C03657=1192.781,332.000,-73.266,-176.346,7.864,148.456
C03658=1192.786,331.751,-73.233,-176.349,7.861,148.456
C03659=1192.790,331.504,-73.202,-176.351,7.857,148.456
C03660=1192.794,331.256,-73.170,-176.354,7.854,148.456
C03661=1192.798,331.008,-73.138,-176.356,7.851,148.455
C03662=1192.803,330.759,-73.107,-176.358,7.849,148.456
C03663=1192.807,330.511,-73.075,-176.360,7.845,148.455
C03664=1192.811,330.264,-73.043,-176.363,7.842,148.455
C03665=1192.815,330.016,-73.011,-176.365,7.839,148.455
C03666=1192.819,329.768,-72.979,-176.367,7.836,148.455
C03667=1192.823,329.520,-72.948,-176.370,7.834,148.455
C03668=1192.827,329.272,-72.916,-176.372,7.830,148.455
C03669=1192.832,329.023,-72.884,-176.375,7.827,148.455
C03670=1192.836,328.776,-72.853,-176.377,7.824,148.455
C03671=1192.840,328.528,-72.821,-176.379,7.821,148.454
C03672=1192.844,328.281,-72.789,-176.382,7.818,148.454
C03673=1192.848,328.033,-72.757,-176.383,7.815,148.454
C03674=1192.853,327.784,-72.726,-176.386,7.812,148.454
C03675=1192.857,327.536,-72.694,-176.388,7.809,148.454
C03676=1192.861,327.288,-72.662,-176.391,7.806,148.454
C03677=1192.865,327.040,-72.632,-176.393,7.802,148.454
C03678=1192.869,326.792,-72.600,-176.395,7.800,148.454
C03679=1192.873,326.545,-72.568,-176.398,7.797,148.454
C03680=1192.878,326.296,-72.537,-176.400,7.794,148.454
C03681=1192.882,326.049,-72.505,-176.403,7.791,148.453
C03682=1192.886,325.801,-72.473,-176.405,7.788,148.453
C03683=1192.891,325.553,-72.443,-176.407,7.785,148.453
C03684=1192.894,325.305,-72.411,-176.410,7.782,148.453
C03685=1192.899,325.057,-72.379,-176.412,7.779,148.453
C03686=1192.903,324.809,-72.348,-176.415,7.776,148.453
C03687=1192.906,324.561,-72.316,-176.417,7.772,148.453
C03688=1192.911,324.313,-72.285,-176.419,7.770,148.453
C03689=1192.915,324.064,-72.253,-176.421,7.767,148.453
C03690=1192.920,323.817,-72.222,-176.424,7.764,148.453
C03691=1192.924,323.568,-72.190,-176.427,7.761,148.453
C03692=1192.928,323.321,-72.159,-176.429,7.757,148.452
C03693=1192.932,323.072,-72.128,-176.432,7.754,148.452
C03694=1192.936,322.825,-72.096,-176.433,7.752,148.452
C03695=1192.940,322.576,-72.065,-176.436,7.749,148.452
C03696=1192.945,322.329,-72.034,-176.438,7.746,148.452
C03697=1192.949,322.081,-72.003,-176.441,7.743,148.452
C03698=1192.953,321.832,-71.972,-176.444,7.740,148.452
C03699=1192.958,321.585,-71.940,-176.445,7.737,148.452
C03700=1192.962,321.336,-71.909,-176.448,7.734,148.452
C03701=1192.966,321.089,-71.878,-176.450,7.731,148.452
C03702=1192.970,320.840,-71.847,-176.453,7.728,148.452
C03703=1192.974,320.593,-71.815,-176.455,7.726,148.452
C03704=1192.978,320.344,-71.784,-176.457,7.722,148.452
C03705=1192.982,320.097,-71.754,-176.460,7.719,148.452
C03706=1192.986,319.849,-71.722,-176.462,7.716,148.451
C03707=1192.990,319.601,-71.691,-176.465,7.713,148.451
C03708=1192.995,319.353,-71.660,-176.467,7.711,148.451
C03709=1192.999,319.105,-71.629,-176.469,7.707,148.451
C03710=1193.003,318.857,-71.598,-176.472,7.704,148.451
C03711=1193.007,318.608,-71.567,-176.475,7.701,148.451
C03712=1193.012,318.360,-71.536,-176.477,7.698,148.451
C03713=1193.016,318.113,-71.504,-176.479,7.696,148.451
C03714=1193.020,317.864,-71.473,-176.482,7.693,148.451
C03715=1193.024,317.616,-71.443,-176.484,7.689,148.451
C03716=1193.029,317.369,-71.412,-176.487,7.686,148.451
C03717=1193.033,317.120,-71.381,-176.489,7.683,148.451
C03718=1193.037,316.873,-71.350,-176.491,7.681,148.451
C03719=1193.041,316.624,-71.319,-176.494,7.678,148.451
C03720=1193.046,316.376,-71.288,-176.496,7.675,148.451
C03721=1193.050,316.128,-71.258,-176.499,7.672,148.451
C03722=1193.054,315.880,-71.227,-176.501,7.669,148.451
C03723=1193.058,315.632,-71.195,-176.504,7.666,148.451
C03724=1193.063,315.384,-71.164,-176.506,7.663,148.450
C03725=1193.067,315.136,-71.133,-176.508,7.660,148.450
C03726=1193.072,314.859,-71.100,-176.511,7.657,148.450
C03727=1193.076,314.583,-71.065,-176.514,7.654,148.450
C03728=1193.081,314.307,-71.031,-176.517,7.651,148.450
C03729=1193.085,314.030,-70.997,-176.519,7.647,148.450
C03730=1193.090,313.782,-70.966,-176.522,7.645,148.450
C03731=1193.094,313.534,-70.935,-176.524,7.642,148.450
C03732=1193.098,313.286,-70.905,-176.527,7.639,148.450
C03733=1193.102,313.038,-70.874,-176.529,7.635,148.450
C03734=1193.107,312.790,-70.843,-176.531,7.633,148.450
C03735=1193.111,312.542,-70.812,-176.534,7.630,148.450
C03736=1193.115,312.293,-70.782,-176.537,7.627,148.450
C03737=1193.119,312.045,-70.751,-176.539,7.624,148.450
C03738=1193.124,311.797,-70.720,-176.542,7.621,148.450
C03739=1193.128,311.550,-70.690,-176.544,7.619,148.450
C03740=1193.132,311.301,-70.659,-176.546,7.616,148.450
C03741=1193.136,311.053,-70.628,-176.549,7.612,148.450
C03742=1193.140,310.805,-70.598,-176.551,7.609,148.450
C03743=1193.145,310.558,-70.567,-176.554,7.607,148.450
C03744=1193.149,310.309,-70.538,-176.556,7.604,148.450
C03745=1193.153,310.061,-70.507,-176.559,7.601,148.450
C03746=1193.158,309.813,-70.476,-176.561,7.598,148.450
C03747=1193.162,309.565,-70.446,-176.563,7.596,148.450
C03748=1193.166,309.317,-70.415,-176.566,7.593,148.450
C03749=1193.170,309.068,-70.384,-176.569,7.590,148.450
C03750=1193.174,308.820,-70.355,-176.571,7.586,148.450
C03751=1193.179,308.572,-70.324,-176.573,7.584,148.450
C03752=1193.183,308.325,-70.294,-176.576,7.581,148.450
C03753=1193.188,308.077,-70.263,-176.579,7.578,148.450
C03754=1193.191,307.828,-70.233,-176.581,7.575,148.450
C03755=1193.196,307.580,-70.202,-176.583,7.573,148.450
C03756=1193.200,307.332,-70.172,-176.586,7.569,148.450
C03757=1193.205,307.083,-70.142,-176.588,7.566,148.450
C03758=1193.208,306.836,-70.112,-176.591,7.563,148.450
C03759=1193.213,306.588,-70.081,-176.593,7.561,148.450
C03760=1193.217,306.339,-70.051,-176.596,7.558,148.450
C03761=1193.221,306.091,-70.021,-176.599,7.555,148.450
C03762=1193.225,305.843,-69.990,-176.601,7.552,148.449
C03763=1193.230,305.595,-69.960,-176.603,7.550,148.449
C03764=1193.234,305.347,-69.930,-176.606,7.547,148.450
C03765=1193.239,305.098,-69.900,-176.608,7.544,148.450
C03766=1193.243,304.851,-69.870,-176.611,7.541,148.450
C03767=1193.247,304.603,-69.839,-176.613,7.539,148.450
C03768=1193.251,304.354,-69.809,-176.616,7.536,148.450
C03769=1193.255,304.106,-69.779,-176.618,7.532,148.449
C03770=1193.260,303.858,-69.749,-176.621,7.529,148.449
C03771=1193.264,303.610,-69.719,-176.623,7.527,148.450
C03772=1193.268,303.361,-69.689,-176.626,7.524,148.450
C03773=1193.272,303.114,-69.659,-176.628,7.521,148.450
C03774=1193.277,302.865,-69.629,-176.631,7.518,148.450
C03775=1193.281,302.618,-69.599,-176.633,7.516,148.450
C03776=1193.285,302.369,-69.569,-176.636,7.513,148.450
C03777=1193.290,302.121,-69.539,-176.639,7.510,148.450
C03778=1193.294,301.873,-69.509,-176.640,7.507,148.450
C03779=1193.298,301.625,-69.479,-176.643,7.504,148.450
C03780=1193.303,301.377,-69.449,-176.646,7.501,148.450
C03781=1193.306,301.128,-69.419,-176.648,7.498,148.450
C03782=1193.311,300.880,-69.389,-176.651,7.496,148.450
C03783=1193.315,300.632,-69.359,-176.653,7.493,148.450
C03784=1193.319,300.383,-69.329,-176.656,7.490,148.450
C03785=1193.324,300.135,-69.300,-176.658,7.488,148.450
C03786=1193.328,299.887,-69.269,-176.661,7.485,148.450
C03787=1193.332,299.639,-69.239,-176.664,7.482,148.450
C03788=1193.337,299.391,-69.210,-176.666,7.479,148.450
C03789=1193.340,299.143,-69.180,-176.668,7.477,148.450
C03790=1193.345,298.894,-69.150,-176.671,7.473,148.450
C03791=1193.350,298.646,-69.120,-176.673,7.470,148.450
C03792=1193.354,298.398,-69.091,-176.676,7.468,148.450
C03793=1193.358,298.150,-69.061,-176.678,7.465,148.450
C03794=1193.363,297.902,-69.031,-176.681,7.462,148.450
C03795=1193.367,297.653,-69.001,-176.684,7.459,148.450
C03796=1193.371,297.405,-68.972,-176.686,7.457,148.450
C03797=1193.375,297.157,-68.942,-176.688,7.454,148.450
C03798=1193.379,296.909,-68.912,-176.691,7.451,148.450
C03799=1193.384,296.661,-68.882,-176.693,7.449,148.450
C03800=1193.388,296.412,-68.853,-176.696,7.446,148.450
C03801=1193.392,296.164,-68.823,-176.699,7.443,148.450
C03802=1193.396,295.916,-68.794,-176.701,7.441,148.450
C03803=1193.401,295.668,-68.765,-176.704,7.438,148.450
C03804=1193.405,295.420,-68.735,-176.706,7.435,148.450
C03805=1193.410,295.172,-68.706,-176.709,7.432,148.450
C03806=1193.414,294.924,-68.675,-176.711,7.429,148.450
C03807=1193.418,294.675,-68.646,-176.714,7.426,148.450
C03808=1193.423,294.427,-68.616,-176.717,7.423,148.450
C03809=1193.427,294.179,-68.587,-176.719,7.421,148.450
C03810=1193.431,293.931,-68.557,-176.721,7.418,148.450
C03811=1193.435,293.682,-68.528,-176.724,7.415,148.450
C03812=1193.439,293.434,-68.498,-176.726,7.413,148.450
C03813=1193.443,293.186,-68.469,-176.729,7.410,148.450
C03814=1193.448,292.938,-68.439,-176.732,7.407,148.450
C03815=1193.452,292.690,-68.410,-176.734,7.405,148.451
C03816=1193.457,292.442,-68.381,-176.737,7.402,148.451
C03817=1193.461,292.193,-68.352,-176.739,7.399,148.451
C03818=1193.465,291.945,-68.323,-176.741,7.397,148.451
C03819=1193.469,291.696,-68.293,-176.744,7.394,148.451
C03820=1193.474,291.448,-68.264,-176.747,7.391,148.451
C03821=1193.478,291.200,-68.234,-176.749,7.388,148.451
C03822=1193.482,290.952,-68.205,-176.752,7.385,148.451
C03823=1193.487,290.704,-68.176,-176.754,7.382,148.451
C03824=1193.491,290.456,-68.146,-176.757,7.380,148.451
C03825=1193.495,290.207,-68.118,-176.759,7.377,148.451
C03826=1193.500,289.959,-68.088,-176.762,7.374,148.451
C03827=1193.504,289.710,-68.059,-176.764,7.372,148.451
C03828=1193.508,289.462,-68.029,-176.767,7.369,148.451
C03829=1193.513,289.214,-68.000,-176.769,7.366,148.451
C03830=1193.517,288.939,-67.968,-176.773,7.363,148.451
C03831=1193.523,288.665,-67.936,-176.775,7.360,148.451
C03832=1193.527,288.391,-67.903,-176.778,7.357,148.451
C03833=1193.531,288.116,-67.871,-176.781,7.354,148.451
C03834=1193.536,287.868,-67.842,-176.784,7.351,148.451
C03835=1193.541,287.619,-67.814,-176.786,7.349,148.452
C03836=1193.545,287.371,-67.784,-176.788,7.346,148.452
C03837=1193.549,287.123,-67.755,-176.791,7.343,148.452
C03838=1193.554,286.875,-67.726,-176.793,7.341,148.452
C03839=1193.558,286.626,-67.697,-176.796,7.338,148.452
C03840=1193.562,286.378,-67.668,-176.799,7.336,148.452
C03841=1193.566,286.130,-67.639,-176.801,7.333,148.452
C03842=1193.570,285.881,-67.610,-176.804,7.330,148.452
C03843=1193.575,285.634,-67.581,-176.806,7.328,148.452
C03844=1193.580,285.385,-67.552,-176.809,7.325,148.452
C03845=1193.584,285.137,-67.523,-176.812,7.322,148.452
C03846=1193.588,284.889,-67.495,-176.814,7.320,148.452
C03847=1193.592,284.640,-67.465,-176.816,7.317,148.452
C03848=1193.597,284.392,-67.437,-176.819,7.314,148.452
C03849=1193.601,284.143,-67.407,-176.821,7.311,148.452
C03850=1193.605,283.895,-67.379,-176.824,7.309,148.453
C03851=1193.609,283.647,-67.350,-176.827,7.307,148.453
C03852=1193.614,283.398,-67.321,-176.829,7.304,148.453
C03853=1193.619,283.151,-67.292,-176.832,7.301,148.453
C03854=1193.622,282.902,-67.264,-176.834,7.298,148.453
C03855=1193.627,282.654,-67.235,-176.837,7.295,148.453
C03856=1193.632,282.406,-67.206,-176.840,7.292,148.453
C03857=1193.636,282.157,-67.177,-176.842,7.290,148.453
C03858=1193.640,281.909,-67.149,-176.844,7.287,148.453
C03859=1193.645,281.661,-67.120,-176.847,7.285,148.453
C03860=1193.649,281.412,-67.091,-176.850,7.282,148.453
C03861=1193.653,281.164,-67.063,-176.852,7.279,148.453
C03862=1193.657,280.916,-67.033,-176.855,7.277,148.453
C03863=1193.662,280.667,-67.005,-176.857,7.274,148.453
C03864=1193.666,280.419,-66.977,-176.859,7.272,148.454
C03865=1193.670,280.171,-66.948,-176.862,7.269,148.454
C03866=1193.674,279.923,-66.919,-176.865,7.266,148.454
C03867=1193.679,279.674,-66.891,-176.868,7.264,148.454
C03868=1193.684,279.426,-66.862,-176.870,7.261,148.454
C03869=1193.687,279.178,-66.833,-176.872,7.259,148.454
C03870=1193.692,278.929,-66.805,-176.875,7.256,148.454
C03871=1193.696,278.681,-66.777,-176.878,7.253,148.454
C03872=1193.700,278.433,-66.747,-176.880,7.251,148.454
C03873=1193.705,278.184,-66.719,-176.883,7.248,148.454
C03874=1193.709,277.936,-66.691,-176.885,7.246,148.454
C03875=1193.714,277.688,-66.663,-176.888,7.243,148.455
C03876=1193.718,277.439,-66.634,-176.891,7.240,148.455
C03877=1193.722,277.191,-66.605,-176.893,7.238,148.455
C03878=1193.726,276.943,-66.577,-176.896,7.235,148.455
C03879=1193.731,276.694,-66.548,-176.898,7.233,148.455
C03880=1193.735,276.446,-66.521,-176.901,7.230,148.455
C03881=1193.740,276.197,-66.492,-176.904,7.227,148.455
C03882=1193.744,275.949,-66.464,-176.906,7.225,148.455
C03883=1193.749,275.700,-66.435,-176.909,7.222,148.455
C03884=1193.752,275.452,-66.407,-176.911,7.220,148.455
C03885=1193.757,275.204,-66.379,-176.914,7.217,148.455
C03886=1193.761,274.956,-66.350,-176.916,7.215,148.456
C03887=1193.766,274.708,-66.322,-176.919,7.212,148.456
C03888=1193.770,274.459,-66.294,-176.921,7.209,148.456
C03889=1193.775,274.211,-66.265,-176.924,7.207,148.456
C03890=1193.779,273.962,-66.237,-176.927,7.204,148.456
C03891=1193.783,273.714,-66.209,-176.929,7.202,148.456
C03892=1193.787,273.465,-66.181,-176.932,7.199,148.456
C03893=1193.792,273.218,-66.153,-176.934,7.197,148.456
C03894=1193.796,272.969,-66.124,-176.937,7.194,148.456
C03895=1193.801,272.721,-66.096,-176.940,7.191,148.456
C03896=1193.805,272.472,-66.069,-176.942,7.189,148.457
C03897=1193.810,272.223,-66.040,-176.944,7.186,148.457
C03898=1193.814,271.975,-66.012,-176.947,7.184,148.457
C03899=1193.819,271.727,-65.984,-176.950,7.181,148.457
C03900=1193.822,271.478,-65.956,-176.952,7.179,148.457
C03901=1193.827,271.230,-65.928,-176.955,7.176,148.457
C03902=1193.831,270.981,-65.899,-176.957,7.174,148.457
C03903=1193.836,270.733,-65.871,-176.960,7.171,148.457
C03904=1193.840,270.486,-65.844,-176.962,7.169,148.457
C03905=1193.845,270.236,-65.816,-176.965,7.166,148.458
C03906=1193.849,269.988,-65.788,-176.968,7.163,148.458
C03907=1193.853,269.740,-65.760,-176.970,7.161,148.458
C03908=1193.858,269.491,-65.731,-176.973,7.158,148.458
C03909=1193.862,269.243,-65.703,-176.975,7.156,148.458
C03910=1193.866,268.994,-65.676,-176.978,7.153,148.458
C03911=1193.871,268.747,-65.648,-176.980,7.151,148.458
C03912=1193.875,268.498,-65.620,-176.983,7.148,148.458
C03913=1193.879,268.250,-65.592,-176.985,7.146,148.458
C03914=1193.884,268.001,-65.564,-176.988,7.143,148.459
C03915=1193.888,267.753,-65.537,-176.991,7.141,148.459
C03916=1193.893,267.504,-65.508,-176.993,7.138,148.459
C03917=1193.897,267.255,-65.481,-176.995,7.136,148.459
C03918=1193.901,267.007,-65.453,-176.999,7.133,148.459
C03919=1193.905,266.759,-65.425,-177.001,7.131,148.459
C03920=1193.910,266.510,-65.398,-177.004,7.128,148.459
C03921=1193.915,266.262,-65.370,-177.006,7.126,148.460
C03922=1193.919,266.014,-65.341,-177.009,7.123,148.460
C03923=1193.923,265.765,-65.314,-177.011,7.121,148.460
C03924=1193.928,265.517,-65.287,-177.014,7.118,148.460
C03925=1193.932,265.268,-65.259,-177.016,7.116,148.460
C03926=1193.936,265.020,-65.231,-177.019,7.113,148.460
C03927=1193.941,264.771,-65.204,-177.021,7.111,148.460
C03928=1193.945,264.523,-65.176,-177.024,7.108,148.460
C03929=1193.950,264.275,-65.148,-177.027,7.106,148.461
C03930=1193.954,264.026,-65.121,-177.029,7.103,148.461
C03931=1193.958,263.778,-65.093,-177.031,7.101,148.461
C03932=1193.963,263.529,-65.065,-177.035,7.098,148.461
C03933=1193.967,263.281,-65.038,-177.037,7.096,148.461
C03934=1193.972,263.007,-65.008,-177.040,7.093,148.461
C03935=1193.977,262.735,-64.977,-177.043,7.090,148.461
C03936=1193.982,262.463,-64.948,-177.045,7.087,148.461
C03937=1193.986,262.189,-64.917,-177.049,7.085,148.462
C03938=1193.991,261.941,-64.889,-177.051,7.082,148.462
C03939=1193.995,261.693,-64.862,-177.054,7.080,148.462
C03940=1193.999,261.444,-64.834,-177.056,7.078,148.462
C03941=1194.004,261.196,-64.807,-177.059,7.075,148.462
C03942=1194.008,260.947,-64.780,-177.061,7.073,148.462
C03943=1194.013,260.699,-64.752,-177.064,7.070,148.462
C03944=1194.017,260.450,-64.725,-177.066,7.068,148.463
C03945=1194.022,260.202,-64.698,-177.070,7.065,148.463
C03946=1194.026,259.954,-64.670,-177.072,7.063,148.463
C03947=1194.031,259.705,-64.643,-177.074,7.060,148.463
C03948=1194.035,259.456,-64.615,-177.077,7.058,148.463
C03949=1194.039,259.208,-64.588,-177.079,7.056,148.463
C03950=1194.044,258.960,-64.561,-177.082,7.053,148.463
C03951=1194.048,258.711,-64.534,-177.085,7.051,148.464
C03952=1194.053,258.463,-64.506,-177.087,7.048,148.464
C03953=1194.057,258.214,-64.478,-177.089,7.046,148.464
C03954=1194.061,257.966,-64.451,-177.093,7.043,148.464
C03955=1194.066,257.717,-64.424,-177.095,7.041,148.464
C03956=1194.071,257.469,-64.397,-177.097,7.038,148.464
C03957=1194.075,257.220,-64.370,-177.100,7.036,148.465
C03958=1194.078,256.972,-64.343,-177.102,7.034,148.465
C03959=1194.083,256.723,-64.315,-177.105,7.031,148.465
C03960=1194.088,256.475,-64.288,-177.108,7.029,148.465
C03961=1194.092,256.226,-64.261,-177.110,7.026,148.465
C03962=1194.097,255.978,-64.234,-177.113,7.024,148.465
C03963=1194.102,255.729,-64.207,-177.116,7.021,148.465
C03964=1194.106,255.480,-64.180,-177.118,7.019,148.466
C03965=1194.110,255.232,-64.153,-177.121,7.016,148.466
C03966=1194.114,254.984,-64.126,-177.123,7.014,148.466
C03967=1194.119,254.736,-64.098,-177.126,7.012,148.466
C03968=1194.123,254.487,-64.071,-177.129,7.009,148.466
C03969=1194.128,254.239,-64.044,-177.131,7.007,148.466
C03970=1194.132,253.991,-64.018,-177.134,7.004,148.467
C03971=1194.136,253.741,-63.990,-177.136,7.002,148.467
C03972=1194.140,253.493,-63.963,-177.139,7.000,148.467
C03973=1194.145,253.244,-63.936,-177.141,6.997,148.467
C03974=1194.150,252.996,-63.909,-177.144,6.995,148.467
C03975=1194.154,252.748,-63.883,-177.147,6.993,148.467
C03976=1194.158,252.499,-63.856,-177.149,6.990,148.468
C03977=1194.163,252.251,-63.829,-177.152,6.988,148.468
C03978=1194.168,252.002,-63.802,-177.154,6.986,148.468
C03979=1194.172,251.753,-63.776,-177.156,6.983,148.468
C03980=1194.177,251.505,-63.749,-177.160,6.981,148.468
C03981=1194.181,251.256,-63.722,-177.162,6.979,148.468
C03982=1194.185,251.008,-63.695,-177.165,6.976,148.469
C03983=1194.189,250.759,-63.668,-177.167,6.974,148.469
C03984=1194.194,250.511,-63.641,-177.170,6.972,148.469
C03985=1194.198,250.262,-63.614,-177.172,6.969,148.469
C03986=1194.202,250.014,-63.587,-177.175,6.967,148.469
C03987=1194.207,249.765,-63.561,-177.178,6.964,148.469
C03988=1194.211,249.517,-63.534,-177.180,6.962,148.470
C03989=1194.216,249.268,-63.507,-177.183,6.960,148.470
C03990=1194.221,249.020,-63.480,-177.185,6.957,148.470
C03991=1194.225,248.771,-63.454,-177.188,6.955,148.470
C03992=1194.230,248.522,-63.428,-177.191,6.952,148.470
C03993=1194.234,248.274,-63.400,-177.193,6.950,148.471
C03994=1194.238,248.026,-63.374,-177.195,6.948,148.471
C03995=1194.243,247.777,-63.347,-177.199,6.946,148.471
C03996=1194.247,247.528,-63.321,-177.201,6.943,148.471
C03997=1194.252,247.280,-63.294,-177.204,6.940,148.471
C03998=1194.256,247.031,-63.267,-177.206,6.939,148.471
C03999=1194.261,246.782,-63.241,-177.208,6.936,148.472
C04000=1194.265,246.534,-63.214,-177.212,6.934,148.472
C04001=1194.269,246.286,-63.188,-177.214,6.932,148.472
C04002=1194.274,246.037,-63.161,-177.216,6.930,148.472
C04003=1194.278,245.788,-63.135,-177.219,6.927,148.472
C04004=1194.283,245.540,-63.108,-177.222,6.925,148.473
C04005=1194.287,245.291,-63.082,-177.224,6.923,148.473
C04006=1194.291,245.043,-63.055,-177.227,6.920,148.473
C04007=1194.296,244.794,-63.029,-177.229,6.918,148.473
C04008=1194.300,244.545,-63.002,-177.232,6.915,148.473
C04009=1194.305,244.298,-62.976,-177.235,6.913,148.473
C04010=1194.310,244.049,-62.950,-177.237,6.911,148.474
C04011=1194.314,243.801,-62.923,-177.240,6.908,148.474
C04012=1194.319,243.551,-62.897,-177.243,6.907,148.474
C04013=1194.323,243.303,-62.871,-177.245,6.904,148.474
C04014=1194.328,243.054,-62.844,-177.248,6.902,148.475
C04015=1194.332,242.806,-62.818,-177.250,6.900,148.475
C04016=1194.337,242.557,-62.791,-177.253,6.898,148.475
C04017=1194.340,242.309,-62.765,-177.255,6.895,148.475
C04018=1194.345,242.060,-62.739,-177.258,6.893,148.475
C04019=1194.349,241.811,-62.712,-177.260,6.891,148.475
C04020=1194.354,241.563,-62.687,-177.263,6.888,148.476
C04021=1194.359,241.314,-62.660,-177.266,6.886,148.476
C04022=1194.363,241.066,-62.634,-177.268,6.884,148.476
C04023=1194.367,240.817,-62.608,-177.271,6.881,148.476
C04024=1194.372,240.569,-62.581,-177.274,6.879,148.476
C04025=1194.376,240.320,-62.555,-177.276,6.877,148.477
C04026=1194.380,240.071,-62.530,-177.279,6.874,148.477
C04027=1194.385,239.823,-62.503,-177.281,6.872,148.477
C04028=1194.390,239.575,-62.477,-177.284,6.870,148.477
C04029=1194.394,239.326,-62.451,-177.287,6.868,148.478
C04030=1194.399,239.077,-62.424,-177.289,6.866,148.478
C04031=1194.403,238.828,-62.399,-177.292,6.864,148.478
C04032=1194.407,238.580,-62.373,-177.294,6.861,148.478
C04033=1194.412,238.332,-62.346,-177.297,6.859,148.478
C04034=1194.417,238.083,-62.320,-177.299,6.857,148.478
C04035=1194.421,237.834,-62.295,-177.302,6.854,148.479
C04036=1194.426,237.585,-62.268,-177.305,6.852,148.479
C04037=1194.430,237.337,-62.242,-177.307,6.850,148.479
C04038=1194.435,237.066,-62.214,-177.310,6.847,148.479
C04039=1194.440,236.794,-62.186,-177.313,6.845,148.480
C04040=1194.444,236.523,-62.157,-177.316,6.843,148.480
C04041=1194.450,236.250,-62.129,-177.319,6.840,148.480
C04042=1194.454,236.002,-62.103,-177.321,6.838,148.480
C04043=1194.458,235.754,-62.077,-177.324,6.836,148.481
C04044=1194.463,235.505,-62.051,-177.327,6.833,148.481
C04045=1194.467,235.256,-62.025,-177.329,6.831,148.481
C04046=1194.472,235.008,-61.999,-177.332,6.829,148.481
C04047=1194.477,234.759,-61.974,-177.334,6.827,148.481
C04048=1194.481,234.510,-61.948,-177.337,6.825,148.482
C04049=1194.485,234.262,-61.922,-177.339,6.822,148.482
C04050=1194.490,234.013,-61.897,-177.342,6.821,148.482
C04051=1194.495,233.764,-61.870,-177.345,6.818,148.482
C04052=1194.499,233.516,-61.844,-177.347,6.816,148.482
C04053=1194.503,233.267,-61.818,-177.350,6.814,148.483
C04054=1194.508,233.019,-61.793,-177.352,6.812,148.483
C04055=1194.512,232.770,-61.767,-177.355,6.809,148.483
C04056=1194.516,232.522,-61.741,-177.358,6.807,148.484
C04057=1194.521,232.274,-61.716,-177.360,6.805,148.484
C04058=1194.525,232.025,-61.690,-177.363,6.802,148.484
C04059=1194.530,231.776,-61.664,-177.366,6.800,148.484
C04060=1194.534,231.527,-61.638,-177.368,6.798,148.484
C04061=1194.540,231.278,-61.613,-177.371,6.797,148.485
C04062=1194.544,231.029,-61.588,-177.374,6.794,148.485
C04063=1194.548,230.780,-61.562,-177.376,6.792,148.485
C04064=1194.553,230.532,-61.537,-177.378,6.790,148.485
C04065=1194.557,230.284,-61.511,-177.381,6.788,148.486
C04066=1194.561,230.035,-61.485,-177.384,6.785,148.486
C04067=1194.566,229.787,-61.460,-177.386,6.783,148.486
C04068=1194.570,229.538,-61.434,-177.389,6.781,148.486
C04069=1194.575,229.289,-61.408,-177.392,6.779,148.487
C04070=1194.579,229.041,-61.383,-177.394,6.776,148.487
C04071=1194.584,228.792,-61.358,-177.397,6.775,148.487
C04072=1194.589,228.543,-61.332,-177.400,6.773,148.487
C04073=1194.593,228.295,-61.307,-177.402,6.770,148.487
C04074=1194.597,228.046,-61.281,-177.405,6.768,148.488
C04075=1194.602,227.798,-61.255,-177.407,6.766,148.488
C04076=1194.607,227.548,-61.230,-177.410,6.764,148.488
C04077=1194.611,227.299,-61.205,-177.413,6.762,148.488
C04078=1194.616,227.051,-61.179,-177.415,6.759,148.489
C04079=1194.620,226.803,-61.154,-177.418,6.757,148.489
C04080=1194.625,226.554,-61.129,-177.421,6.755,148.489
C04081=1194.629,226.305,-61.103,-177.423,6.753,148.489
C04082=1194.633,226.056,-61.077,-177.426,6.751,148.490
C04083=1194.638,225.808,-61.053,-177.429,6.749,148.490
C04084=1194.642,225.559,-61.028,-177.431,6.747,148.490
C04085=1194.647,225.311,-61.002,-177.433,6.745,148.490
C04086=1194.651,225.061,-60.977,-177.437,6.742,148.491
C04087=1194.656,224.813,-60.952,-177.439,6.740,148.491
C04088=1194.660,224.565,-60.926,-177.441,6.738,148.491
C04089=1194.666,224.316,-60.901,-177.444,6.736,148.491
C04090=1194.670,224.067,-60.876,-177.447,6.733,148.491
C04091=1194.674,223.818,-60.850,-177.449,6.732,148.492
C04092=1194.678,223.570,-60.826,-177.452,6.730,148.492
C04093=1194.683,223.321,-60.800,-177.455,6.728,148.492
C04094=1194.688,223.072,-60.775,-177.457,6.726,148.493
C04095=1194.692,222.824,-60.750,-177.460,6.723,148.493
C04096=1194.697,222.575,-60.725,-177.463,6.721,148.493
C04097=1194.701,222.326,-60.700,-177.465,6.719,148.493
C04098=1194.706,222.078,-60.675,-177.468,6.717,148.494
C04099=1194.710,221.829,-60.649,-177.471,6.715,148.494
C04100=1194.715,221.580,-60.625,-177.473,6.713,148.494
C04101=1194.719,221.331,-60.599,-177.476,6.711,148.494
C04102=1194.724,221.083,-60.575,-177.478,6.709,148.495
C04103=1194.728,220.834,-60.549,-177.481,6.707,148.495
C04104=1194.733,220.585,-60.524,-177.484,6.704,148.495
C04105=1194.737,220.336,-60.499,-177.486,6.702,148.495
C04106=1194.742,220.088,-60.475,-177.489,6.700,148.496
C04107=1194.746,219.839,-60.449,-177.491,6.698,148.496
C04108=1194.751,219.591,-60.424,-177.494,6.696,148.496
C04109=1194.755,219.341,-60.400,-177.497,6.694,148.497
C04110=1194.760,219.093,-60.374,-177.500,6.692,148.497
C04111=1194.765,218.845,-60.350,-177.502,6.690,148.497
C04112=1194.769,218.595,-60.325,-177.504,6.688,148.497
C04113=1194.773,218.347,-60.300,-177.507,6.686,148.498
C04114=1194.778,218.098,-60.275,-177.510,6.684,148.498
C04115=1194.783,217.849,-60.250,-177.512,6.681,148.498
C04116=1194.787,217.601,-60.225,-177.515,6.680,148.498
C04117=1194.792,217.352,-60.200,-177.518,6.678,148.499
C04118=1194.795,217.103,-60.176,-177.520,6.676,148.499
C04119=1194.800,216.855,-60.150,-177.523,6.673,148.499
C04120=1194.805,216.606,-60.126,-177.526,6.671,148.499
C04121=1194.809,216.357,-60.101,-177.528,6.669,148.500
C04122=1194.814,216.108,-60.077,-177.531,6.667,148.500
C04123=1194.819,215.859,-60.051,-177.533,6.665,148.500
C04124=1194.823,215.611,-60.027,-177.536,6.663,148.501
C04125=1194.828,215.362,-60.002,-177.539,6.661,148.501
C04126=1194.832,215.113,-59.978,-177.542,6.659,148.501
C04127=1194.837,214.864,-59.953,-177.544,6.657,148.501
C04128=1194.841,214.617,-59.928,-177.547,6.655,148.502
C04129=1194.846,214.367,-59.903,-177.549,6.653,148.502
C04130=1194.851,214.119,-59.879,-177.552,6.651,148.502
C04131=1194.855,213.870,-59.855,-177.555,6.648,148.502
C04132=1194.860,213.621,-59.829,-177.557,6.647,148.503
C04133=1194.864,213.372,-59.805,-177.560,6.645,148.503
C04134=1194.869,213.123,-59.780,-177.563,6.643,148.503
C04135=1194.873,212.874,-59.756,-177.565,6.641,148.504
C04136=1194.878,212.626,-59.731,-177.568,6.638,148.504
C04137=1194.882,212.377,-59.706,-177.571,6.636,148.504
C04138=1194.887,212.129,-59.682,-177.573,6.635,148.505
C04139=1194.891,211.880,-59.658,-177.576,6.633,148.505
C04140=1194.896,211.631,-59.633,-177.578,6.631,148.505
C04141=1194.900,211.382,-59.609,-177.581,6.629,148.505
C04142=1194.905,211.112,-59.582,-177.584,6.626,148.506
C04143=1194.911,210.841,-59.556,-177.587,6.624,148.506
C04144=1194.915,210.570,-59.529,-177.590,6.622,148.506
C04145=1194.920,210.301,-59.503,-177.592,6.620,148.507
C04146=1194.925,210.052,-59.478,-177.595,6.618,148.507
C04147=1194.929,209.803,-59.454,-177.598,6.616,148.507
C04148=1194.934,209.554,-59.429,-177.600,6.613,148.507
C04149=1194.938,209.306,-59.405,-177.603,6.611,148.508
C04150=1194.943,209.057,-59.380,-177.606,6.610,148.508
C04151=1194.948,208.808,-59.356,-177.608,6.608,148.508
C04152=1194.952,208.559,-59.332,-177.611,6.606,148.509
C04153=1194.957,208.310,-59.308,-177.613,6.604,148.509
C04154=1194.961,208.062,-59.284,-177.616,6.602,148.509
C04155=1194.966,207.813,-59.260,-177.619,6.600,148.510
C04156=1194.970,207.564,-59.235,-177.622,6.598,148.510
C04157=1194.975,207.315,-59.210,-177.624,6.596,148.510
C04158=1194.979,207.067,-59.186,-177.627,6.594,148.510
C04159=1194.984,206.818,-59.162,-177.629,6.592,148.511
C04160=1194.989,206.569,-59.138,-177.632,6.590,148.511
C04161=1194.993,206.320,-59.114,-177.635,6.588,148.511
C04162=1194.998,206.071,-59.089,-177.637,6.586,148.512
C04163=1195.002,205.823,-59.065,-177.640,6.585,148.512
C04164=1195.007,205.574,-59.042,-177.643,6.582,148.512
C04165=1195.012,205.325,-59.017,-177.645,6.580,148.512
C04166=1195.016,205.076,-58.993,-177.648,6.578,148.513
C04167=1195.020,204.827,-58.969,-177.651,6.576,148.513
C04168=1195.025,204.579,-58.945,-177.653,6.574,148.513
C04169=1195.030,204.330,-58.921,-177.656,6.572,148.514
C04170=1195.034,204.081,-58.897,-177.658,6.570,148.514
C04171=1195.039,203.832,-58.873,-177.661,6.569,148.514
C04172=1195.043,203.583,-58.849,-177.663,6.567,148.515
C04173=1195.048,203.335,-58.824,-177.667,6.564,148.515
C04174=1195.053,203.086,-58.801,-177.669,6.562,148.515
C04175=1195.057,202.837,-58.777,-177.672,6.560,148.516
C04176=1195.062,202.588,-58.753,-177.675,6.559,148.516
C04177=1195.066,202.340,-58.729,-177.677,6.556,148.516
C04178=1195.071,202.090,-58.704,-177.679,6.555,148.516
C04179=1195.075,201.841,-58.681,-177.682,6.553,148.517
C04180=1195.080,201.593,-58.657,-177.685,6.551,148.517
C04181=1195.085,201.344,-58.633,-177.687,6.549,148.517
C04182=1195.089,201.095,-58.609,-177.690,6.547,148.518
C04183=1195.093,200.847,-58.585,-177.693,6.546,148.518
C04184=1195.098,200.598,-58.562,-177.695,6.543,148.518
C04185=1195.103,200.349,-58.537,-177.698,6.541,148.519
C04186=1195.108,200.100,-58.514,-177.701,6.539,148.519
C04187=1195.112,199.851,-58.489,-177.703,6.537,148.519
C04188=1195.116,199.602,-58.466,-177.706,6.535,148.520
C04189=1195.121,199.354,-58.442,-177.709,6.534,148.520
C04190=1195.125,199.105,-58.419,-177.711,6.532,148.520
C04191=1195.130,198.856,-58.395,-177.714,6.530,148.521
C04192=1195.135,198.607,-58.371,-177.716,6.528,148.521
C04193=1195.139,198.358,-58.348,-177.719,6.526,148.521
C04194=1195.144,198.110,-58.324,-177.721,6.524,148.521
C04195=1195.148,197.861,-58.300,-177.724,6.522,148.522
C04196=1195.153,197.612,-58.276,-177.727,6.521,148.522
C04197=1195.158,197.363,-58.252,-177.729,6.519,148.522
C04198=1195.163,197.114,-58.229,-177.732,6.517,148.523
C04199=1195.167,196.865,-58.205,-177.735,6.514,148.523
C04200=1195.172,196.616,-58.182,-177.737,6.512,148.523
C04201=1195.177,196.367,-58.158,-177.740,6.510,148.524
C04202=1195.181,196.119,-58.134,-177.743,6.509,148.524
C04203=1195.186,195.870,-58.111,-177.745,6.507,148.524
C04204=1195.190,195.621,-58.087,-177.748,6.505,148.525
C04205=1195.195,195.373,-58.063,-177.751,6.503,148.525
C04206=1195.200,195.124,-58.040,-177.753,6.501,148.525
C04207=1195.204,194.874,-58.017,-177.756,6.500,148.526
C04208=1195.208,194.626,-57.994,-177.759,6.498,148.526
C04209=1195.213,194.377,-57.970,-177.761,6.496,148.526
C04210=1195.217,194.128,-57.946,-177.764,6.494,148.527
C04211=1195.222,193.879,-57.923,-177.766,6.492,148.527
C04212=1195.227,193.630,-57.900,-177.769,6.490,148.527
C04213=1195.231,193.382,-57.876,-177.772,6.488,148.528
C04214=1195.236,193.133,-57.852,-177.774,6.487,148.528
C04215=1195.240,192.884,-57.829,-177.777,6.485,148.528
C04216=1195.245,192.635,-57.806,-177.780,6.483,148.529
C04217=1195.250,192.386,-57.782,-177.782,6.481,148.529
C04218=1195.255,192.137,-57.759,-177.785,6.479,148.529
C04219=1195.259,191.888,-57.735,-177.788,6.478,148.530
C04220=1195.263,191.640,-57.712,-177.790,6.476,148.530
C04221=1195.268,191.390,-57.689,-177.793,6.474,148.530
C04222=1195.272,191.141,-57.665,-177.796,6.472,148.531
C04223=1195.277,190.892,-57.642,-177.798,6.470,148.531
C04224=1195.282,190.644,-57.619,-177.800,6.468,148.531
C04225=1195.287,190.395,-57.596,-177.803,6.466,148.532
C04226=1195.292,190.146,-57.572,-177.806,6.465,148.532
C04227=1195.296,189.897,-57.549,-177.808,6.463,148.532
C04228=1195.300,189.648,-57.526,-177.811,6.461,148.533
C04229=1195.305,189.399,-57.503,-177.814,6.459,148.533
C04230=1195.310,189.150,-57.479,-177.816,6.457,148.533
C04231=1195.315,188.901,-57.456,-177.819,6.456,148.534
C04232=1195.318,188.652,-57.433,-177.822,6.454,148.534
C04233=1195.324,188.404,-57.410,-177.824,6.452,148.534
C04234=1195.328,188.155,-57.387,-177.827,6.450,148.535
C04235=1195.333,187.906,-57.364,-177.830,6.448,148.535
C04236=1195.337,187.657,-57.341,-177.832,6.447,148.535
C04237=1195.342,187.408,-57.317,-177.835,6.445,148.536
C04238=1195.347,187.159,-57.294,-177.838,6.443,148.536
C04239=1195.351,186.910,-57.271,-177.840,6.441,148.536
C04240=1195.356,186.662,-57.248,-177.843,6.439,148.537
C04241=1195.360,186.413,-57.225,-177.846,6.438,148.537
C04242=1195.365,186.164,-57.202,-177.848,6.436,148.538
C04243=1195.369,185.915,-57.179,-177.851,6.434,148.538
C04244=1195.374,185.666,-57.156,-177.853,6.432,148.538
C04245=1195.379,185.417,-57.133,-177.856,6.430,148.538
C04246=1195.383,185.147,-57.108,-177.859,6.428,148.539
C04247=1195.388,184.878,-57.083,-177.862,6.426,148.539
C04248=1195.394,184.608,-57.058,-177.865,6.424,148.540
C04249=1195.398,184.339,-57.033,-177.867,6.422,148.540
C04250=1195.404,184.090,-57.011,-177.870,6.420,148.540
C04251=1195.409,183.841,-56.988,-177.873,6.419,148.541
C04252=1195.413,183.592,-56.965,-177.875,6.417,148.541
C04253=1195.417,183.343,-56.941,-177.878,6.415,148.541
C04254=1195.421,183.094,-56.919,-177.881,6.413,148.542
C04255=1195.427,182.846,-56.896,-177.883,6.411,148.542
C04256=1195.432,182.596,-56.873,-177.886,6.410,148.542
C04257=1195.436,182.348,-56.850,-177.889,6.408,148.543
C04258=1195.441,182.098,-56.828,-177.891,6.406,148.543
C04259=1195.445,181.850,-56.805,-177.894,6.404,148.544
C04260=1195.450,181.601,-56.782,-177.897,6.402,148.544
C04261=1195.454,181.352,-56.760,-177.899,6.401,148.544
C04262=1195.459,181.103,-56.736,-177.902,6.399,148.545
C04263=1195.464,180.854,-56.713,-177.905,6.397,148.545
C04264=1195.468,180.605,-56.691,-177.907,6.395,148.545
C04265=1195.473,180.356,-56.668,-177.910,6.394,148.546
C04266=1195.477,180.107,-56.645,-177.912,6.392,148.546
C04267=1195.483,179.858,-56.623,-177.915,6.391,148.546
C04268=1195.487,179.610,-56.600,-177.918,6.389,148.547
C04269=1195.492,179.360,-56.578,-177.920,6.387,148.547
C04270=1195.496,179.112,-56.555,-177.923,6.385,148.548
C04271=1195.501,178.863,-56.532,-177.926,6.383,148.548
C04272=1195.505,178.614,-56.510,-177.928,6.382,148.548
C04273=1195.510,178.365,-56.487,-177.931,6.380,148.549
C04274=1195.515,178.116,-56.465,-177.934,6.378,148.549
C04275=1195.519,177.867,-56.442,-177.936,6.376,148.549
C04276=1195.524,177.618,-56.420,-177.939,6.375,148.550
C04277=1195.528,177.369,-56.397,-177.942,6.373,148.550
C04278=1195.533,177.120,-56.374,-177.944,6.371,148.550
C04279=1195.538,176.872,-56.352,-177.947,6.369,148.551
C04280=1195.543,176.622,-56.329,-177.949,6.368,148.551
C04281=1195.547,176.373,-56.306,-177.952,6.366,148.552
C04282=1195.552,176.125,-56.285,-177.954,6.365,148.552
C04283=1195.556,175.876,-56.261,-177.957,6.363,148.552
C04284=1195.561,175.626,-56.239,-177.960,6.361,148.553
C04285=1195.566,175.377,-56.217,-177.962,6.359,148.553
C04286=1195.570,175.129,-56.194,-177.965,6.357,148.553
C04287=1195.574,174.879,-56.172,-177.968,6.356,148.554
C04288=1195.580,174.631,-56.149,-177.970,6.354,148.554
C04289=1195.584,174.382,-56.127,-177.973,6.352,148.555
C04290=1195.590,174.133,-56.105,-177.976,6.351,148.555
C04291=1195.594,173.884,-56.082,-177.978,6.350,148.555
C04292=1195.598,173.635,-56.060,-177.981,6.348,148.556
C04293=1195.603,173.386,-56.038,-177.984,6.346,148.556
C04294=1195.607,173.137,-56.015,-177.986,6.344,148.556
C04295=1195.612,172.888,-55.993,-177.989,6.342,148.557
C04296=1195.617,172.639,-55.971,-177.992,6.341,148.557
C04297=1195.621,172.390,-55.948,-177.994,6.339,148.558
C04298=1195.626,172.141,-55.926,-177.997,6.337,148.558
C04299=1195.630,171.892,-55.904,-178.000,6.335,148.558
C04300=1195.636,171.643,-55.882,-178.002,6.334,148.559
C04301=1195.640,171.394,-55.859,-178.004,6.332,148.559
C04302=1195.645,171.146,-55.838,-178.007,6.331,148.559
C04303=1195.649,170.896,-55.816,-178.010,6.329,148.560
C04304=1195.655,170.647,-55.793,-178.012,6.327,148.560
C04305=1195.659,170.398,-55.771,-178.016,6.326,148.561
C04306=1195.663,170.149,-55.748,-178.018,6.324,148.561
C04307=1195.668,169.901,-55.727,-178.021,6.322,148.561
C04308=1195.673,169.651,-55.704,-178.023,6.321,148.562
C04309=1195.678,169.402,-55.682,-178.026,6.319,148.562
C04310=1195.682,169.153,-55.660,-178.028,6.317,148.563
C04311=1195.687,168.904,-55.639,-178.031,6.316,148.563
C04312=1195.691,168.655,-55.617,-178.034,6.314,148.563
C04313=1195.696,168.407,-55.594,-178.036,6.312,148.564
C04314=1195.701,168.157,-55.572,-178.039,6.310,148.564
C04315=1195.706,167.909,-55.550,-178.042,6.309,148.564
C04316=1195.710,167.659,-55.528,-178.044,6.308,148.565
C04317=1195.715,167.411,-55.506,-178.047,6.306,148.565
C04318=1195.719,167.162,-55.484,-178.050,6.304,148.566
C04319=1195.725,166.913,-55.462,-178.052,6.303,148.566
C04320=1195.729,166.663,-55.440,-178.055,6.301,148.566
C04321=1195.734,166.415,-55.418,-178.058,6.299,148.567
C04322=1195.739,166.166,-55.396,-178.060,6.298,148.567
C04323=1195.743,165.917,-55.374,-178.062,6.296,148.568
C04324=1195.748,165.668,-55.353,-178.065,6.294,148.568
C04325=1195.752,165.419,-55.331,-178.068,6.293,148.568
C04326=1195.757,165.170,-55.309,-178.070,6.291,148.569
C04327=1195.761,164.921,-55.287,-178.074,6.289,148.569
C04328=1195.767,164.672,-55.265,-178.076,6.288,148.570
C04329=1195.771,164.422,-55.243,-178.078,6.287,148.570
C04330=1195.776,164.174,-55.221,-178.081,6.285,148.570
C04331=1195.781,163.925,-55.199,-178.084,6.283,148.571
C04332=1195.785,163.676,-55.177,-178.086,6.281,148.571
C04333=1195.790,163.427,-55.156,-178.089,6.279,148.571
C04334=1195.794,163.177,-55.134,-178.092,6.278,148.572
C04335=1195.799,162.928,-55.113,-178.094,6.277,148.572
C04336=1195.804,162.679,-55.090,-178.097,6.275,148.573
C04337=1195.808,162.430,-55.069,-178.100,6.273,148.573
C04338=1195.813,162.182,-55.047,-178.102,6.272,148.574
C04339=1195.818,161.933,-55.025,-178.105,6.270,148.574
C04340=1195.822,161.684,-55.003,-178.107,6.269,148.574
C04341=1195.828,161.435,-54.982,-178.110,6.267,148.575
C04342=1195.832,161.185,-54.960,-178.112,6.265,148.575
C04343=1195.837,160.937,-54.939,-178.116,6.264,148.576
C04344=1195.841,160.687,-54.917,-178.118,6.262,148.576
C04345=1195.846,160.439,-54.895,-178.121,6.260,148.576
C04346=1195.851,160.189,-54.874,-178.123,6.259,148.577
C04347=1195.855,159.940,-54.852,-178.126,6.258,148.577
C04348=1195.859,159.692,-54.831,-178.128,6.256,148.578
C04349=1195.865,159.442,-54.810,-178.131,6.254,148.578
C04350=1195.870,159.174,-54.786,-178.134,6.253,148.579
C04351=1195.875,158.905,-54.763,-178.137,6.251,148.579
C04352=1195.880,158.635,-54.740,-178.140,6.249,148.579
C04353=1195.884,158.367,-54.716,-178.143,6.248,148.580
C04354=1195.890,158.118,-54.695,-178.145,6.246,148.580
C04355=1195.894,157.868,-54.673,-178.148,6.245,148.581
C04356=1195.899,157.620,-54.651,-178.150,6.243,148.581
C04357=1195.904,157.370,-54.631,-178.153,6.241,148.581
C04358=1195.908,157.121,-54.608,-178.156,6.239,148.582
C04359=1195.913,156.872,-54.587,-178.159,6.238,148.582
C04360=1195.918,156.623,-54.566,-178.161,6.237,148.583
C04361=1195.922,156.374,-54.544,-178.164,6.235,148.583
C04362=1195.927,156.125,-54.523,-178.166,6.234,148.583
C04363=1195.932,155.876,-54.502,-178.169,6.232,148.584
C04364=1195.937,155.627,-54.481,-178.171,6.231,148.584
C04365=1195.941,155.378,-54.459,-178.174,6.229,148.585
C04366=1195.945,155.129,-54.438,-178.177,6.228,148.585
C04367=1195.951,154.880,-54.417,-178.180,6.226,148.586
C04368=1195.955,154.631,-54.395,-178.182,6.224,148.586
C04369=1195.960,154.381,-54.374,-178.184,6.223,148.586
C04370=1195.965,154.133,-54.352,-178.187,6.221,148.587
C04371=1195.969,153.884,-54.332,-178.190,6.220,148.587
C04372=1195.974,153.635,-54.310,-178.193,6.218,148.588
C04373=1195.979,153.385,-54.289,-178.195,6.217,148.588
C04374=1195.984,153.137,-54.267,-178.198,6.215,148.588
C04375=1195.988,152.888,-54.247,-178.200,6.214,148.589
C04376=1195.993,152.638,-54.226,-178.203,6.212,148.589
C04377=1195.998,152.390,-54.204,-178.206,6.211,148.590
C04378=1196.003,152.140,-54.183,-178.208,6.209,148.590
C04379=1196.007,151.891,-54.161,-178.211,6.208,148.591
C04380=1196.012,151.642,-54.140,-178.214,6.206,148.591
C04381=1196.017,151.393,-54.120,-178.216,6.205,148.592
C04382=1196.021,151.145,-54.098,-178.219,6.203,148.592
C04383=1196.026,150.895,-54.077,-178.222,6.202,148.592
C04384=1196.031,150.646,-54.055,-178.224,6.200,148.593
C04385=1196.035,150.397,-54.035,-178.226,6.199,148.593
C04386=1196.040,150.148,-54.014,-178.230,6.197,148.594
C04387=1196.045,149.899,-53.992,-178.232,6.196,148.594
C04388=1196.049,149.649,-53.972,-178.235,6.194,148.594
C04389=1196.054,149.400,-53.951,-178.237,6.193,148.595
C04390=1196.059,149.152,-53.929,-178.240,6.191,148.595
C04391=1196.064,148.903,-53.909,-178.243,6.190,148.596
C04392=1196.069,148.653,-53.888,-178.246,6.188,148.596
C04393=1196.074,148.404,-53.867,-178.248,6.187,148.597
C04394=1196.078,148.156,-53.846,-178.250,6.185,148.597
C04395=1196.083,147.906,-53.824,-178.253,6.183,148.597
C04396=1196.087,147.657,-53.804,-178.256,6.182,148.598
C04397=1196.092,147.408,-53.783,-178.258,6.181,148.598
C04398=1196.096,147.159,-53.762,-178.261,6.179,148.599
C04399=1196.102,146.910,-53.741,-178.264,6.177,148.599
C04400=1196.107,146.661,-53.720,-178.266,6.177,148.600
C04401=1196.111,146.412,-53.700,-178.269,6.175,148.600
C04402=1196.116,146.163,-53.679,-178.272,6.173,148.601
C04403=1196.121,145.914,-53.658,-178.274,6.172,148.601
C04404=1196.125,145.664,-53.636,-178.277,6.171,148.602
C04405=1196.129,145.415,-53.616,-178.280,6.169,148.602
C04406=1196.135,145.166,-53.595,-178.282,6.167,148.602
C04407=1196.139,144.917,-53.574,-178.284,6.166,148.603
C04408=1196.144,144.668,-53.553,-178.287,6.165,148.603
C04409=1196.149,144.419,-53.533,-178.290,6.163,148.604
C04410=1196.154,144.170,-53.512,-178.292,6.162,148.604
C04411=1196.158,143.921,-53.492,-178.295,6.160,148.604
C04412=1196.163,143.671,-53.471,-178.298,6.159,148.605
C04413=1196.168,143.423,-53.450,-178.301,6.157,148.605
C04414=1196.173,143.174,-53.429,-178.303,6.156,148.606
C04415=1196.177,142.925,-53.408,-178.306,6.155,148.606
C04416=1196.182,142.676,-53.387,-178.308,6.153,148.607
C04417=1196.187,142.427,-53.367,-178.311,6.152,148.607
C04418=1196.191,142.178,-53.347,-178.314,6.150,148.608
C04419=1196.196,141.929,-53.326,-178.316,6.149,148.608
C04420=1196.201,141.680,-53.305,-178.318,6.148,148.608
C04421=1196.205,141.430,-53.284,-178.322,6.146,148.609
C04422=1196.210,141.181,-53.264,-178.324,6.144,148.609
C04423=1196.214,140.932,-53.243,-178.326,6.144,148.610
C04424=1196.220,140.682,-53.223,-178.329,6.142,148.610
C04425=1196.224,140.433,-53.203,-178.332,6.140,148.611
C04426=1196.229,140.184,-53.182,-178.335,6.139,148.611
C04427=1196.234,139.935,-53.161,-178.337,6.138,148.612
C04428=1196.238,139.686,-53.141,-178.340,6.136,148.612
C04429=1196.243,139.436,-53.120,-178.343,6.134,148.613
C04430=1196.248,139.188,-53.100,-178.345,6.133,148.613
C04431=1196.253,138.939,-53.080,-178.348,6.132,148.613
C04432=1196.258,138.690,-53.059,-178.351,6.130,148.614
C04433=1196.263,138.441,-53.038,-178.353,6.129,148.614
C04434=1196.267,138.191,-53.019,-178.356,6.128,148.615
C04435=1196.272,137.942,-52.998,-178.358,6.126,148.615
C04436=1196.277,137.693,-52.977,-178.361,6.125,148.616
C04437=1196.281,137.444,-52.957,-178.364,6.123,148.616
C04438=1196.287,137.195,-52.936,-178.366,6.122,148.617
C04439=1196.291,136.945,-52.916,-178.369,6.121,148.617
C04440=1196.296,136.697,-52.896,-178.372,6.119,148.618
C04441=1196.300,136.448,-52.875,-178.374,6.118,148.618
C04442=1196.305,136.198,-52.855,-178.376,6.116,148.618
C04443=1196.310,135.949,-52.834,-178.380,6.115,148.619
C04444=1196.314,135.700,-52.815,-178.382,6.114,148.619
C04445=1196.320,135.451,-52.794,-178.384,6.112,148.620
C04446=1196.324,135.202,-52.773,-178.388,6.111,148.620
C04447=1196.329,134.953,-52.754,-178.390,6.110,148.621
C04448=1196.334,134.704,-52.734,-178.392,6.108,148.621
C04449=1196.338,134.455,-52.713,-178.396,6.107,148.622
C04450=1196.343,134.206,-52.692,-178.398,6.106,148.622
C04451=1196.348,133.956,-52.673,-178.400,6.104,148.623
C04452=1196.353,133.707,-52.652,-178.403,6.102,148.623
C04453=1196.357,133.457,-52.632,-178.406,6.102,148.624
C04454=1196.363,133.189,-52.610,-178.408,6.100,148.624
C04455=1196.368,132.921,-52.589,-178.412,6.099,148.625
C04456=1196.373,132.652,-52.567,-178.414,6.097,148.625
C04457=1196.378,132.384,-52.546,-178.417,6.096,148.626
C04458=1196.383,132.134,-52.525,-178.420,6.094,148.626
C04459=1196.388,131.885,-52.505,-178.422,6.093,148.626
C04460=1196.392,131.636,-52.485,-178.425,6.092,148.627
C04461=1196.398,131.387,-52.465,-178.428,6.090,148.627
C04462=1196.402,131.138,-52.445,-178.430,6.088,148.628
C04463=1196.407,130.889,-52.424,-178.433,6.088,148.628
C04464=1196.411,130.639,-52.405,-178.436,6.086,148.629
C04465=1196.416,130.390,-52.384,-178.438,6.085,148.629
C04466=1196.421,130.141,-52.364,-178.441,6.084,148.630
C04467=1196.426,129.892,-52.344,-178.443,6.082,148.630
C04468=1196.431,129.643,-52.325,-178.446,6.081,148.631
C04469=1196.435,129.394,-52.304,-178.449,6.080,148.631
C04470=1196.440,129.144,-52.285,-178.451,6.079,148.632
C04471=1196.445,128.895,-52.264,-178.454,6.077,148.632
C04472=1196.450,128.646,-52.245,-178.457,6.076,148.633
C04473=1196.454,128.397,-52.224,-178.459,6.075,148.633
C04474=1196.459,128.148,-52.205,-178.462,6.073,148.633
C04475=1196.464,127.898,-52.185,-178.464,6.072,148.634
C04476=1196.468,127.649,-52.165,-178.467,6.070,148.634
C04477=1196.474,127.401,-52.146,-178.470,6.069,148.635
C04478=1196.478,127.152,-52.125,-178.472,6.068,148.635
C04479=1196.483,126.902,-52.105,-178.475,6.066,148.636
C04480=1196.488,126.652,-52.086,-178.477,6.065,148.636
C04481=1196.493,126.404,-52.066,-178.480,6.064,148.637
C04482=1196.497,126.155,-52.046,-178.483,6.062,148.637
C04483=1196.502,125.905,-52.027,-178.485,6.061,148.638
C04484=1196.506,125.656,-52.006,-178.488,6.060,148.638
C04485=1196.512,125.407,-51.987,-178.490,6.059,148.639
C04486=1196.517,125.158,-51.967,-178.493,6.057,148.639
C04487=1196.521,124.909,-51.947,-178.496,6.057,148.640
C04488=1196.526,124.659,-51.927,-178.498,6.055,148.640
C04489=1196.531,124.410,-51.908,-178.501,6.053,148.641
C04490=1196.536,124.161,-51.887,-178.504,6.052,148.641
C04491=1196.540,123.912,-51.868,-178.506,6.051,148.642
C04492=1196.546,123.663,-51.849,-178.509,6.050,148.642
C04493=1196.550,123.413,-51.829,-178.512,6.048,148.643
C04494=1196.555,123.164,-51.809,-178.514,6.047,148.643
C04495=1196.559,122.916,-51.790,-178.517,6.046,148.644
C04496=1196.564,122.666,-51.770,-178.520,6.044,148.644
C04497=1196.569,122.417,-51.751,-178.522,6.044,148.645
C04498=1196.574,122.167,-51.731,-178.525,6.042,148.645
C04499=1196.579,121.919,-51.711,-178.527,6.041,148.645
C04500=1196.583,121.669,-51.691,-178.530,6.039,148.646
C04501=1196.588,121.420,-51.672,-178.532,6.039,148.647
C04502=1196.594,121.171,-51.652,-178.535,6.037,148.647
C04503=1196.598,120.922,-51.633,-178.538,6.035,148.648
C04504=1196.603,120.673,-51.614,-178.540,6.034,148.648
C04505=1196.607,120.424,-51.594,-178.543,6.033,148.649
C04506=1196.612,120.174,-51.574,-178.546,6.032,148.649
C04507=1196.617,119.925,-51.555,-178.548,6.030,148.649
C04508=1196.622,119.676,-51.535,-178.551,6.030,148.650
C04509=1196.626,119.427,-51.516,-178.554,6.028,148.650
C04510=1196.631,119.178,-51.497,-178.556,6.027,148.651
C04511=1196.636,118.928,-51.477,-178.559,6.026,148.651
C04512=1196.641,118.679,-51.457,-178.561,6.025,148.652
C04513=1196.646,118.430,-51.438,-178.564,6.023,148.652
C04514=1196.650,118.180,-51.419,-178.566,6.022,148.653
C04515=1196.656,117.932,-51.400,-178.569,6.021,148.653
C04516=1196.660,117.682,-51.380,-178.572,6.019,148.654
C04517=1196.665,117.432,-51.360,-178.574,6.018,148.654
C04518=1196.670,117.184,-51.342,-178.578,6.017,148.655
C04519=1196.674,116.934,-51.322,-178.580,6.016,148.655
C04520=1196.680,116.685,-51.303,-178.582,6.014,148.656
C04521=1196.685,116.436,-51.283,-178.585,6.014,148.656
C04522=1196.689,116.187,-51.264,-178.588,6.012,148.657
C04523=1196.694,115.938,-51.245,-178.590,6.011,148.657
C04524=1196.699,115.688,-51.225,-178.593,6.009,148.658
C04525=1196.703,115.440,-51.206,-178.595,6.009,148.658
C04526=1196.708,115.190,-51.187,-178.598,6.007,148.659
C04527=1196.713,114.941,-51.167,-178.600,6.006,148.659
C04528=1196.718,114.692,-51.148,-178.604,6.005,148.660
C04529=1196.723,114.443,-51.129,-178.606,6.004,148.660
C04530=1196.727,114.193,-51.109,-178.609,6.002,148.661
C04531=1196.733,113.944,-51.091,-178.611,6.002,148.661
C04532=1196.737,113.695,-51.072,-178.614,6.000,148.662
C04533=1196.742,113.446,-51.052,-178.616,5.999,148.662
C04534=1196.746,113.197,-51.033,-178.619,5.997,148.663
C04535=1196.752,112.948,-51.014,-178.622,5.997,148.663
C04536=1196.757,112.698,-50.994,-178.624,5.995,148.664
C04537=1196.761,112.448,-50.976,-178.627,5.994,148.664
C04538=1196.766,112.199,-50.957,-178.630,5.993,148.665
C04539=1196.771,111.950,-50.937,-178.632,5.992,148.665
C04540=1196.776,111.701,-50.918,-178.635,5.990,148.666
C04541=1196.780,111.452,-50.899,-178.637,5.989,148.666
C04542=1196.785,111.203,-50.881,-178.640,5.988,148.667
C04543=1196.791,110.954,-50.861,-178.642,5.987,148.667
C04544=1196.795,110.704,-50.842,-178.646,5.986,148.668
C04545=1196.800,110.456,-50.823,-178.648,5.985,148.668
C04546=1196.805,110.205,-50.804,-178.650,5.983,148.669
C04547=1196.810,109.957,-50.786,-178.653,5.982,148.669
C04548=1196.814,109.707,-50.766,-178.656,5.981,148.670
C04549=1196.819,109.458,-50.748,-178.658,5.980,148.670
C04550=1196.824,109.208,-50.728,-178.661,5.978,148.671
C04551=1196.829,108.960,-50.710,-178.664,5.978,148.672
C04552=1196.834,108.710,-50.691,-178.666,5.976,148.672
C04553=1196.838,108.461,-50.672,-178.669,5.975,148.673
C04554=1196.843,108.212,-50.652,-178.672,5.974,148.673
C04555=1196.848,107.962,-50.634,-178.674,5.973,148.673
C04556=1196.853,107.714,-50.615,-178.677,5.971,148.674
C04557=1196.857,107.464,-50.596,-178.679,5.970,148.674
C04558=1196.863,107.196,-50.576,-178.682,5.969,148.675
C04559=1196.868,106.927,-50.555,-178.685,5.968,148.676
C04560=1196.873,106.659,-50.535,-178.688,5.967,148.676
C04561=1196.879,106.391,-50.515,-178.691,5.965,148.677
C04562=1196.883,106.141,-50.496,-178.693,5.964,148.677
C04563=1196.888,105.892,-50.477,-178.696,5.963,148.678
C04564=1196.893,105.643,-50.459,-178.698,5.962,148.678
C04565=1196.898,105.393,-50.439,-178.701,5.962,148.679
C04566=1196.903,105.144,-50.421,-178.704,5.960,148.679
C04567=1196.908,104.895,-50.402,-178.706,5.959,148.680
C04568=1196.912,104.646,-50.384,-178.709,5.957,148.680
C04569=1196.917,104.397,-50.365,-178.712,5.957,148.681
C04570=1196.922,104.147,-50.346,-178.714,5.955,148.681
C04571=1196.927,103.898,-50.327,-178.717,5.955,148.682
C04572=1196.932,103.649,-50.309,-178.720,5.953,148.682
C04573=1196.936,103.399,-50.290,-178.722,5.952,148.683
C04574=1196.941,103.150,-50.272,-178.724,5.951,148.683
C04575=1196.946,102.901,-50.252,-178.727,5.950,148.684
C04576=1196.951,102.652,-50.234,-178.730,5.949,148.685
C04577=1196.956,102.403,-50.216,-178.732,5.947,148.685
C04578=1196.961,102.153,-50.197,-178.735,5.947,148.686
C04579=1196.965,101.904,-50.179,-178.738,5.945,148.686
C04580=1196.970,101.655,-50.160,-178.740,5.944,148.687
C04581=1196.975,101.405,-50.141,-178.743,5.943,148.687
C04582=1196.980,101.156,-50.123,-178.746,5.942,148.688
C04583=1196.985,100.907,-50.104,-178.748,5.941,148.688
C04584=1196.990,100.658,-50.086,-178.751,5.940,148.689
C04585=1196.994,100.408,-50.067,-178.753,5.939,148.689
C04586=1196.999,100.159,-50.049,-178.756,5.937,148.690
C04587=1197.004,99.910,-50.031,-178.758,5.936,148.690
C04588=1197.009,99.660,-50.011,-178.761,5.936,148.691
C04589=1197.014,99.411,-49.993,-178.764,5.934,148.691
C04590=1197.019,99.162,-49.975,-178.766,5.934,148.692
C04591=1197.024,98.913,-49.956,-178.769,5.932,148.692
C04592=1197.028,98.663,-49.937,-178.772,5.931,148.693
C04593=1197.033,98.414,-49.919,-178.774,5.929,148.693
C04594=1197.038,98.165,-49.901,-178.777,5.929,148.694
C04595=1197.043,97.915,-49.882,-178.779,5.928,148.694
C04596=1197.048,97.666,-49.864,-178.782,5.927,148.695
C04597=1197.053,97.417,-49.846,-178.784,5.926,148.696
C04598=1197.058,97.168,-49.828,-178.788,5.924,148.696
C04599=1197.062,96.918,-49.810,-178.790,5.923,148.697
C04600=1197.067,96.669,-49.790,-178.792,5.923,148.697
C04601=1197.072,96.420,-49.772,-178.795,5.921,148.698
C04602=1197.077,96.171,-49.754,-178.798,5.920,148.698
C04603=1197.081,95.921,-49.736,-178.800,5.919,148.699
C04604=1197.086,95.672,-49.718,-178.803,5.918,148.699
C04605=1197.091,95.423,-49.700,-178.805,5.917,148.700
C04606=1197.097,95.174,-49.681,-178.808,5.916,148.700
C04607=1197.102,94.925,-49.663,-178.810,5.915,148.701
C04608=1197.106,94.675,-49.644,-178.814,5.914,148.701
C04609=1197.111,94.426,-49.626,-178.816,5.913,148.702
C04610=1197.116,94.176,-49.608,-178.818,5.912,148.703
C04611=1197.121,93.927,-49.590,-178.821,5.910,148.703
C04612=1197.125,93.678,-49.572,-178.824,5.910,148.704
C04613=1197.131,93.428,-49.553,-178.826,5.909,148.704
C04614=1197.135,93.179,-49.536,-178.829,5.907,148.705
C04615=1197.140,92.930,-49.517,-178.832,5.907,148.705
C04616=1197.145,92.681,-49.499,-178.834,5.905,148.706
C04617=1197.150,92.432,-49.481,-178.837,5.905,148.706
C04618=1197.155,92.183,-49.463,-178.839,5.904,148.707
C04619=1197.159,91.933,-49.445,-178.842,5.902,148.707
C04620=1197.164,91.684,-49.427,-178.844,5.901,148.708
C04621=1197.169,91.434,-49.409,-178.847,5.901,148.709
C04622=1197.174,91.185,-49.391,-178.850,5.899,148.709
C04623=1197.179,90.936,-49.373,-178.852,5.898,148.710
C04624=1197.184,90.687,-49.355,-178.855,5.897,148.710
C04625=1197.189,90.438,-49.337,-178.858,5.896,148.711
C04626=1197.193,90.188,-49.318,-178.860,5.895,148.711
C04627=1197.198,89.939,-49.300,-178.863,5.894,148.712
C04628=1197.203,89.689,-49.283,-178.866,5.893,148.712
C04629=1197.209,89.439,-49.264,-178.868,5.892,148.713
C04630=1197.214,89.190,-49.247,-178.871,5.891,148.713
C04631=1197.218,88.941,-49.229,-178.873,5.890,148.714
C04632=1197.223,88.692,-49.211,-178.876,5.889,148.714
C04633=1197.228,88.443,-49.193,-178.879,5.888,148.715
C04634=1197.232,88.194,-49.175,-178.881,5.887,148.716
C04635=1197.237,87.944,-49.157,-178.883,5.886,148.716
C04636=1197.242,87.695,-49.139,-178.886,5.885,148.717
C04637=1197.247,87.445,-49.121,-178.889,5.884,148.717
C04638=1197.252,87.196,-49.104,-178.892,5.883,148.718
C04639=1197.257,86.947,-49.086,-178.894,5.882,148.718
C04640=1197.262,86.697,-49.068,-178.897,5.881,148.719
C04641=1197.267,86.448,-49.050,-178.900,5.880,148.719
C04642=1197.271,86.199,-49.032,-178.902,5.879,148.720
C04643=1197.277,85.949,-49.014,-178.905,5.878,148.721
C04644=1197.282,85.700,-48.996,-178.907,5.877,148.721
C04645=1197.287,85.451,-48.978,-178.910,5.876,148.722
C04646=1197.291,85.202,-48.960,-178.912,5.875,148.722
C04647=1197.296,84.953,-48.943,-178.915,5.874,148.723
C04648=1197.301,84.703,-48.926,-178.918,5.873,148.723
C04649=1197.306,84.454,-48.908,-178.920,5.872,148.724
C04650=1197.311,84.205,-48.890,-178.923,5.871,148.724
C04651=1197.315,83.955,-48.872,-178.925,5.870,148.725
C04652=1197.320,83.705,-48.854,-178.928,5.869,148.725
C04653=1197.325,83.456,-48.836,-178.931,5.868,148.726
C04654=1197.330,83.207,-48.818,-178.933,5.867,148.727
C04655=1197.334,82.957,-48.802,-178.936,5.866,148.727
C04656=1197.339,82.708,-48.784,-178.938,5.866,148.728
C04657=1197.344,82.459,-48.766,-178.941,5.864,148.728
C04658=1197.350,82.209,-48.748,-178.943,5.863,148.729
C04659=1197.354,81.960,-48.730,-178.946,5.863,148.729
C04660=1197.359,81.711,-48.712,-178.949,5.861,148.730
C04661=1197.364,81.461,-48.696,-178.951,5.860,148.730
C04662=1197.370,81.194,-48.677,-178.955,5.859,148.731
C04663=1197.375,80.925,-48.658,-178.957,5.858,148.732
C04664=1197.380,80.656,-48.639,-178.959,5.858,148.732
C04665=1197.385,80.388,-48.620,-178.962,5.856,148.733
C04666=1197.390,80.138,-48.602,-178.965,5.856,148.733
C04667=1197.395,79.889,-48.585,-178.968,5.854,148.734
C04668=1197.400,79.640,-48.567,-178.970,5.853,148.735
C04669=1197.405,79.390,-48.550,-178.973,5.853,148.735
C04670=1197.410,79.141,-48.532,-178.975,5.852,148.736
C04671=1197.415,78.893,-48.515,-178.978,5.851,148.736
C04672=1197.420,78.643,-48.498,-178.981,5.850,148.737
C04673=1197.425,78.394,-48.480,-178.983,5.849,148.737
C04674=1197.430,78.144,-48.463,-178.986,5.847,148.738
C04675=1197.434,77.895,-48.445,-178.989,5.847,148.738
C04676=1197.439,77.645,-48.428,-178.991,5.846,148.739
C04677=1197.444,77.396,-48.410,-178.994,5.844,148.739
C04678=1197.449,77.147,-48.393,-178.996,5.844,148.740
C04679=1197.454,76.897,-48.375,-178.999,5.843,148.741
C04680=1197.459,76.648,-48.358,-179.001,5.842,148.741
C04681=1197.463,76.398,-48.341,-179.004,5.841,148.742
C04682=1197.468,76.149,-48.323,-179.007,5.840,148.742
C04683=1197.474,75.900,-48.306,-179.009,5.840,148.743
C04684=1197.478,75.651,-48.289,-179.011,5.839,148.743
C04685=1197.483,75.401,-48.272,-179.015,5.837,148.744
C04686=1197.488,75.152,-48.254,-179.017,5.837,148.745
C04687=1197.493,74.903,-48.237,-179.019,5.836,148.745
C04688=1197.498,74.653,-48.220,-179.023,5.834,148.746
C04689=1197.503,74.404,-48.202,-179.025,5.834,148.746
C04690=1197.507,74.154,-48.185,-179.027,5.833,148.747
C04691=1197.513,73.905,-48.168,-179.030,5.832,148.748
C04692=1197.517,73.656,-48.151,-179.033,5.831,148.748
C04693=1197.523,73.406,-48.134,-179.035,5.830,148.749
C04694=1197.528,73.157,-48.116,-179.038,5.830,148.749
C04695=1197.532,72.908,-48.099,-179.040,5.829,148.750
C04696=1197.537,72.658,-48.082,-179.043,5.827,148.750
C04697=1197.542,72.408,-48.065,-179.045,5.826,148.751
C04698=1197.547,72.160,-48.048,-179.048,5.826,148.751
C04699=1197.552,71.910,-48.031,-179.051,5.825,148.752
C04700=1197.557,71.661,-48.014,-179.053,5.824,148.753
C04701=1197.562,71.411,-47.996,-179.056,5.823,148.753
C04702=1197.566,71.162,-47.979,-179.059,5.823,148.754
C04703=1197.572,70.913,-47.962,-179.061,5.822,148.754
C04704=1197.577,70.663,-47.945,-179.064,5.820,148.755
C04705=1197.582,70.414,-47.928,-179.066,5.819,148.755
C04706=1197.586,70.165,-47.911,-179.069,5.819,148.756
C04707=1197.591,69.915,-47.893,-179.071,5.818,148.757
C04708=1197.596,69.666,-47.877,-179.074,5.817,148.757
C04709=1197.602,69.416,-47.860,-179.077,5.816,148.758
C04710=1197.606,69.167,-47.843,-179.079,5.815,148.758
C04711=1197.611,68.918,-47.825,-179.082,5.815,148.759
C04712=1197.615,68.668,-47.809,-179.085,5.813,148.760
C04713=1197.621,68.419,-47.792,-179.087,5.812,148.760
C04714=1197.626,68.170,-47.775,-179.089,5.812,148.761
C04715=1197.631,67.920,-47.758,-179.092,5.811,148.761
C04716=1197.635,67.670,-47.741,-179.095,5.809,148.762
C04717=1197.641,67.422,-47.725,-179.097,5.809,148.762
C04718=1197.646,67.172,-47.707,-179.100,5.808,148.763
C04719=1197.650,66.923,-47.690,-179.102,5.807,148.763
C04720=1197.655,66.673,-47.673,-179.105,5.807,148.764
C04721=1197.660,66.424,-47.657,-179.108,5.806,148.765
C04722=1197.665,66.175,-47.639,-179.110,5.805,148.765
C04723=1197.670,65.925,-47.623,-179.113,5.804,148.766
C04724=1197.674,65.676,-47.606,-179.115,5.804,148.767
C04725=1197.680,65.426,-47.589,-179.118,5.802,148.767
C04726=1197.685,65.177,-47.572,-179.121,5.801,148.768
C04727=1197.689,64.928,-47.556,-179.123,5.800,148.768
C04728=1197.695,64.678,-47.539,-179.126,5.800,148.769
C04729=1197.699,64.429,-47.522,-179.128,5.799,148.769
C04730=1197.705,64.179,-47.505,-179.131,5.798,148.770
C04731=1197.709,63.930,-47.488,-179.134,5.797,148.770
C04732=1197.714,63.681,-47.472,-179.136,5.796,148.771
C04733=1197.719,63.431,-47.455,-179.138,5.796,148.772
C04734=1197.724,63.182,-47.438,-179.141,5.795,148.772
C04735=1197.729,62.933,-47.422,-179.144,5.794,148.773
C04736=1197.734,62.683,-47.404,-179.146,5.793,148.773
C04737=1197.739,62.434,-47.388,-179.149,5.792,148.774
C04738=1197.744,62.185,-47.371,-179.152,5.792,148.775
C04739=1197.749,61.935,-47.354,-179.154,5.791,148.775
C04740=1197.753,61.685,-47.337,-179.157,5.789,148.776
C04741=1197.759,61.436,-47.322,-179.160,5.789,148.776
C04742=1197.763,61.187,-47.305,-179.162,5.788,148.777
C04743=1197.769,60.937,-47.288,-179.164,5.787,148.778
C04744=1197.774,60.688,-47.272,-179.167,5.787,148.778
C04745=1197.778,60.439,-47.255,-179.170,5.785,148.779
C04746=1197.784,60.189,-47.238,-179.172,5.785,148.779
C04747=1197.788,59.940,-47.221,-179.175,5.784,148.780
C04748=1197.793,59.690,-47.205,-179.177,5.783,148.780
C04749=1197.798,59.441,-47.189,-179.180,5.783,148.781
C04750=1197.804,59.191,-47.172,-179.183,5.781,148.782
C04751=1197.808,58.942,-47.155,-179.185,5.780,148.782
C04752=1197.813,58.693,-47.139,-179.188,5.780,148.783
C04753=1197.818,58.444,-47.122,-179.190,5.779,148.783
C04754=1197.823,58.194,-47.107,-179.193,5.778,148.784
C04755=1197.828,57.944,-47.089,-179.195,5.778,148.785
C04756=1197.833,57.695,-47.073,-179.198,5.777,148.785
C04757=1197.838,57.446,-47.056,-179.201,5.776,148.786
C04758=1197.843,57.196,-47.040,-179.203,5.775,148.786
C04759=1197.848,56.947,-47.024,-179.206,5.775,148.787
C04760=1197.853,56.697,-47.007,-179.208,5.774,148.787
C04761=1197.857,56.448,-46.990,-179.211,5.772,148.788
C04762=1197.863,56.198,-46.975,-179.214,5.772,148.789
C04763=1197.867,55.949,-46.958,-179.216,5.771,148.789
C04764=1197.872,55.700,-46.942,-179.219,5.770,148.790
C04765=1197.877,55.450,-46.926,-179.221,5.770,148.791
C04766=1197.883,55.182,-46.907,-179.224,5.769,148.791
C04767=1197.889,54.913,-46.890,-179.227,5.768,148.792
C04768=1197.893,54.645,-46.872,-179.229,5.767,148.792
C04769=1197.899,54.376,-46.855,-179.232,5.766,148.793
C04770=1197.903,54.127,-46.839,-179.235,5.765,148.794
C04771=1197.909,53.878,-46.823,-179.238,5.765,148.794
C04772=1197.914,53.628,-46.806,-179.240,5.764,148.795
C04773=1197.919,53.379,-46.789,-179.243,5.763,148.795
C04774=1197.924,53.129,-46.773,-179.245,5.763,148.796
C04775=1197.929,52.880,-46.757,-179.248,5.762,148.797
C04776=1197.933,52.631,-46.741,-179.251,5.760,148.797
C04777=1197.939,52.381,-46.725,-179.253,5.760,148.798
C04778=1197.943,52.132,-46.708,-179.256,5.759,148.799
C04779=1197.949,51.882,-46.693,-179.258,5.758,148.799
C04780=1197.953,51.633,-46.676,-179.261,5.758,148.800
C04781=1197.958,51.383,-46.660,-179.263,5.757,148.800
C04782=1197.963,51.134,-46.644,-179.265,5.756,148.801
C04783=1197.968,50.885,-46.628,-179.269,5.755,148.801
C04784=1197.973,50.635,-46.611,-179.271,5.755,148.802
C04785=1197.978,50.386,-46.596,-179.274,5.754,148.803
C04786=1197.983,50.136,-46.579,-179.276,5.753,148.803
C04787=1197.988,49.887,-46.564,-179.279,5.753,148.804
C04788=1197.992,49.637,-46.547,-179.281,5.752,148.805
C04789=1197.998,49.388,-46.531,-179.283,5.751,148.805
C04790=1198.002,49.138,-46.515,-179.286,5.751,148.806
C04791=1198.008,48.889,-46.499,-179.289,5.749,148.806
C04792=1198.012,48.639,-46.482,-179.291,5.748,148.807
C04793=1198.018,48.390,-46.467,-179.294,5.748,148.807
C04794=1198.023,48.141,-46.451,-179.297,5.747,148.808
C04795=1198.027,47.891,-46.435,-179.299,5.747,148.809
C04796=1198.033,47.642,-46.419,-179.302,5.746,148.809
C04797=1198.037,47.392,-46.402,-179.304,5.745,148.810
C04798=1198.043,47.143,-46.387,-179.307,5.745,148.811
C04799=1198.047,46.893,-46.370,-179.310,5.743,148.811
C04800=1198.053,46.644,-46.355,-179.312,5.743,148.812
C04801=1198.058,46.395,-46.339,-179.315,5.742,148.812
C04802=1198.062,46.145,-46.322,-179.317,5.742,148.813
C04803=1198.068,45.896,-46.307,-179.320,5.741,148.813
C04804=1198.072,45.646,-46.291,-179.322,5.740,148.814
C04805=1198.077,45.397,-46.275,-179.325,5.740,148.815
C04806=1198.082,45.148,-46.259,-179.327,5.739,148.815
C04807=1198.087,44.898,-46.243,-179.330,5.738,148.816
C04808=1198.092,44.649,-46.227,-179.333,5.737,148.817
C04809=1198.097,44.399,-46.211,-179.336,5.736,148.817
C04810=1198.102,44.149,-46.196,-179.338,5.735,148.818
C04811=1198.107,43.901,-46.179,-179.340,5.735,148.818
C04812=1198.112,43.650,-46.163,-179.343,5.734,148.819
C04813=1198.117,43.401,-46.148,-179.345,5.734,148.819
C04814=1198.122,43.152,-46.133,-179.348,5.733,148.820
C04815=1198.127,42.902,-46.116,-179.350,5.732,148.821
C04816=1198.132,42.653,-46.101,-179.353,5.732,148.821
C04817=1198.137,42.403,-46.085,-179.355,5.731,148.822
C04818=1198.142,42.154,-46.069,-179.358,5.731,148.823
C04819=1198.147,41.905,-46.053,-179.361,5.729,148.823
C04820=1198.151,41.655,-46.037,-179.364,5.729,148.824
C04821=1198.157,41.406,-46.022,-179.366,5.728,148.824
C04822=1198.162,41.156,-46.006,-179.368,5.727,148.825
C04823=1198.167,40.906,-45.990,-179.371,5.727,148.826
C04824=1198.172,40.657,-45.975,-179.373,5.726,148.826
C04825=1198.177,40.408,-45.959,-179.376,5.725,148.827
C04826=1198.182,40.159,-45.943,-179.379,5.725,148.828
C04827=1198.187,39.909,-45.927,-179.381,5.724,148.828
C04828=1198.192,39.660,-45.912,-179.383,5.723,148.829
C04829=1198.197,39.410,-45.897,-179.386,5.723,148.829
C04830=1198.202,39.160,-45.881,-179.389,5.722,148.830
C04831=1198.207,38.911,-45.865,-179.392,5.721,148.831
C04832=1198.212,38.662,-45.850,-179.394,5.720,148.831
C04833=1198.216,38.412,-45.834,-179.397,5.720,148.832
C04834=1198.222,38.163,-45.818,-179.399,5.719,148.832
C04835=1198.227,37.913,-45.802,-179.402,5.719,148.833
C04836=1198.232,37.664,-45.787,-179.404,5.718,148.834
C04837=1198.236,37.414,-45.771,-179.407,5.717,148.834
C04838=1198.242,37.165,-45.756,-179.409,5.717,148.835
C04839=1198.247,36.916,-45.741,-179.412,5.716,148.836
C04840=1198.252,36.666,-45.725,-179.414,5.715,148.836
C04841=1198.257,36.416,-45.709,-179.417,5.715,148.837
C04842=1198.262,36.167,-45.694,-179.419,5.714,148.837
C04843=1198.267,35.918,-45.679,-179.422,5.713,148.838
C04844=1198.272,35.668,-45.663,-179.424,5.713,148.839
C04845=1198.277,35.418,-45.647,-179.427,5.712,148.839
C04846=1198.282,35.169,-45.632,-179.430,5.712,148.840
C04847=1198.287,34.920,-45.617,-179.432,5.710,148.840
C04848=1198.292,34.671,-45.602,-179.435,5.709,148.841
C04849=1198.296,34.420,-45.586,-179.438,5.709,148.842
C04850=1198.302,34.171,-45.570,-179.440,5.708,148.842
C04851=1198.306,33.922,-45.555,-179.442,5.708,148.843
C04852=1198.312,33.673,-45.540,-179.445,5.707,148.843
C04853=1198.317,33.423,-45.524,-179.448,5.707,148.844
C04854=1198.322,33.173,-45.509,-179.450,5.706,148.845
C04855=1198.327,32.923,-45.494,-179.452,5.705,148.845
C04856=1198.332,32.674,-45.479,-179.455,5.705,148.846
C04857=1198.337,32.425,-45.463,-179.458,5.704,148.847
C04858=1198.342,32.175,-45.448,-179.460,5.704,148.847
C04859=1198.346,31.926,-45.432,-179.463,5.703,148.848
C04860=1198.352,31.676,-45.417,-179.465,5.702,148.848
C04861=1198.356,31.427,-45.402,-179.468,5.702,148.849
C04862=1198.362,31.177,-45.387,-179.470,5.701,148.850
C04863=1198.367,30.928,-45.372,-179.473,5.701,148.850
C04864=1198.372,30.679,-45.356,-179.475,5.700,148.851
C04865=1198.376,30.429,-45.341,-179.478,5.699,148.852
C04866=1198.382,30.179,-45.325,-179.481,5.699,148.852
C04867=1198.387,29.930,-45.310,-179.483,5.698,148.853
C04868=1198.392,29.680,-45.295,-179.485,5.697,148.853
C04869=1198.397,29.431,-45.280,-179.488,5.697,148.854
C04870=1198.402,29.163,-45.263,-179.491,5.695,148.855
C04871=1198.408,28.894,-45.247,-179.494,5.695,148.855
C04872=1198.413,28.625,-45.231,-179.496,5.694,148.856
C04873=1198.419,28.356,-45.214,-179.499,5.694,148.857
C04874=1198.424,28.107,-45.200,-179.502,5.693,148.857
C04875=1198.428,27.857,-45.184,-179.504,5.693,148.858
C04876=1198.433,27.607,-45.169,-179.507,5.692,148.859
C04877=1198.438,27.358,-45.153,-179.509,5.691,148.859
C04878=1198.443,27.108,-45.139,-179.512,5.691,148.860
C04879=1198.449,26.859,-45.124,-179.515,5.690,148.861
C04880=1198.453,26.610,-45.109,-179.517,5.690,148.861
C04881=1198.459,26.360,-45.094,-179.519,5.689,148.862
C04882=1198.464,26.111,-45.079,-179.522,5.689,148.862
C04883=1198.468,25.862,-45.064,-179.525,5.688,148.863
C04884=1198.474,25.611,-45.049,-179.527,5.687,148.864
C04885=1198.478,25.362,-45.034,-179.529,5.687,148.864
C04886=1198.484,25.112,-45.018,-179.532,5.686,148.865
C04887=1198.489,24.863,-45.004,-179.535,5.686,148.866
C04888=1198.493,24.614,-44.989,-179.537,5.685,148.866
C04889=1198.499,24.364,-44.973,-179.539,5.684,148.867
C04890=1198.504,24.115,-44.959,-179.542,5.684,148.867
C04891=1198.509,23.865,-44.943,-179.545,5.683,148.868
C04892=1198.514,23.615,-44.929,-179.547,5.683,148.869
C04893=1198.519,23.366,-44.914,-179.550,5.682,148.869
C04894=1198.524,23.116,-44.899,-179.552,5.681,148.870
C04895=1198.529,22.867,-44.884,-179.555,5.681,148.871
C04896=1198.534,22.618,-44.869,-179.558,5.680,148.871
C04897=1198.539,22.368,-44.854,-179.560,5.680,148.872
C04898=1198.544,22.119,-44.839,-179.562,5.679,148.872
C04899=1198.549,21.869,-44.825,-179.565,5.678,148.873
C04900=1198.554,21.620,-44.809,-179.568,5.678,148.874
C04901=1198.559,21.370,-44.795,-179.570,5.677,148.874
C04902=1198.564,21.121,-44.780,-179.572,5.677,148.875
C04903=1198.569,20.871,-44.765,-179.575,5.676,148.876
C04904=1198.574,20.622,-44.750,-179.578,5.675,148.876
C04905=1198.579,20.372,-44.736,-179.580,5.675,148.877
C04906=1198.584,20.123,-44.720,-179.583,5.674,148.878
C04907=1198.589,19.873,-44.706,-179.585,5.674,148.878
C04908=1198.594,19.624,-44.691,-179.588,5.673,148.879
C04909=1198.600,19.374,-44.676,-179.590,5.673,148.879
C04910=1198.605,19.124,-44.662,-179.593,5.672,148.880
C04911=1198.609,18.875,-44.647,-179.595,5.671,148.881
C04912=1198.614,18.626,-44.633,-179.598,5.671,148.881
C04913=1198.620,18.376,-44.617,-179.601,5.670,148.882
C04914=1198.625,18.126,-44.603,-179.603,5.670,148.883
C04915=1198.629,17.877,-44.588,-179.606,5.669,148.883
C04916=1198.634,17.628,-44.574,-179.608,5.668,148.884
C04917=1198.640,17.378,-44.559,-179.611,5.668,148.884
C04918=1198.645,17.129,-44.544,-179.613,5.667,148.885
C04919=1198.650,16.879,-44.529,-179.616,5.667,148.886
C04920=1198.655,16.629,-44.515,-179.619,5.666,148.886
C04921=1198.659,16.380,-44.500,-179.621,5.665,148.887
C04922=1198.665,16.130,-44.485,-179.623,5.665,148.888
C04923=1198.670,15.880,-44.471,-179.626,5.665,148.888
C04924=1198.674,15.631,-44.456,-179.628,5.665,148.889
C04925=1198.679,15.381,-44.442,-179.631,5.664,148.890
C04926=1198.684,15.132,-44.427,-179.633,5.663,148.890
C04927=1198.690,14.882,-44.412,-179.636,5.663,148.891
C04928=1198.695,14.633,-44.398,-179.638,5.662,148.891
C04929=1198.700,14.384,-44.384,-179.641,5.662,148.892
C04930=1198.705,14.135,-44.369,-179.644,5.661,148.893
C04931=1198.710,13.885,-44.354,-179.646,5.660,148.893
C04932=1198.715,13.635,-44.340,-179.648,5.660,148.894
C04933=1198.720,13.385,-44.326,-179.651,5.659,148.895
C04934=1198.725,13.136,-44.310,-179.654,5.659,148.895
C04935=1198.730,12.886,-44.296,-179.656,5.658,148.896
C04936=1198.735,12.637,-44.282,-179.658,5.658,148.896
C04937=1198.740,12.387,-44.267,-179.661,5.657,148.897
C04938=1198.746,12.138,-44.253,-179.664,5.657,148.898
C04939=1198.750,11.889,-44.239,-179.666,5.656,148.899
C04940=1198.755,11.639,-44.224,-179.669,5.656,148.899
C04941=1198.760,11.389,-44.210,-179.671,5.656,148.900
C04942=1198.765,11.140,-44.196,-179.673,5.655,148.900
C04943=1198.771,10.890,-44.181,-179.676,5.655,148.901
C04944=1198.776,10.640,-44.167,-179.679,5.654,148.902
C04945=1198.781,10.392,-44.152,-179.681,5.654,148.902
C04946=1198.786,10.142,-44.138,-179.683,5.653,148.903
C04947=1198.791,9.892,-44.123,-179.686,5.652,148.904
C04948=1198.796,9.642,-44.109,-179.689,5.652,148.904
C04949=1198.801,9.393,-44.095,-179.691,5.651,148.905
C04950=1198.806,9.143,-44.081,-179.694,5.651,148.906
C04951=1198.811,8.893,-44.066,-179.696,5.650,148.906
C04952=1198.816,8.644,-44.052,-179.699,5.649,148.907
C04953=1198.821,8.395,-44.037,-179.702,5.649,148.907
C04954=1198.826,8.145,-44.023,-179.704,5.648,148.908
C04955=1198.831,7.896,-44.009,-179.706,5.649,148.909
C04956=1198.836,7.646,-43.994,-179.708,5.648,148.909
C04957=1198.841,7.397,-43.981,-179.711,5.647,148.910
C04958=1198.846,7.147,-43.966,-179.714,5.647,148.911
C04959=1198.851,6.898,-43.952,-179.716,5.646,148.911
C04960=1198.856,6.648,-43.938,-179.719,5.646,148.912
C04961=1198.861,6.398,-43.923,-179.721,5.645,148.912
C04962=1198.867,6.149,-43.910,-179.724,5.644,148.913
C04963=1198.872,5.899,-43.895,-179.726,5.644,148.914
C04964=1198.877,5.650,-43.881,-179.729,5.643,148.915
C04965=1198.882,5.400,-43.867,-179.732,5.643,148.915
C04966=1198.887,5.150,-43.852,-179.733,5.643,148.916
C04967=1198.892,4.901,-43.839,-179.736,5.642,148.916
C04968=1198.897,4.652,-43.824,-179.739,5.642,148.917
C04969=1198.902,4.402,-43.810,-179.741,5.641,148.918
C04970=1198.906,4.153,-43.796,-179.744,5.641,148.918
C04971=1198.912,3.904,-43.782,-179.747,5.640,148.919
C04972=1198.917,3.654,-43.768,-179.749,5.640,148.920
C04973=1198.922,3.404,-43.754,-179.751,5.639,148.920
C04974=1198.927,3.135,-43.739,-179.754,5.639,148.921
C04975=1198.933,2.866,-43.724,-179.757,5.638,148.922
C04976=1198.939,2.597,-43.709,-179.759,5.638,148.922
C04977=1198.944,2.328,-43.694,-179.762,5.637,148.923
C04978=1198.949,2.078,-43.679,-179.765,5.637,148.924
C04979=1198.954,1.828,-43.666,-179.767,5.636,148.924
C04980=1198.960,1.579,-43.652,-179.770,5.636,148.925
C04981=1198.964,1.329,-43.637,-179.773,5.635,148.926
C04982=1198.969,1.079,-43.623,-179.774,5.635,148.926
C04983=1198.974,0.831,-43.610,-179.777,5.635,148.927
C04984=1198.979,0.581,-43.596,-179.780,5.634,148.928
C04985=1198.984,0.331,-43.581,-179.782,5.634,148.928
C04986=1198.990,0.082,-43.568,-179.785,5.633,148.929
C04987=1198.995,-0.168,-43.554,-179.787,5.632,148.929
C04988=1199.000,-0.418,-43.540,-179.790,5.632,148.930
C04989=1199.004,-0.667,-43.526,-179.792,5.631,148.931
C04990=1199.010,-0.916,-43.512,-179.794,5.632,148.931
C04991=1199.015,-1.167,-43.498,-179.797,5.631,148.932
C04992=1199.020,-1.416,-43.484,-179.800,5.631,148.933
C04993=1199.025,-1.665,-43.470,-179.802,5.630,148.933
C04994=1199.030,-1.915,-43.457,-179.805,5.629,148.934
C04995=1199.035,-2.165,-43.443,-179.807,5.629,148.935
C04996=1199.040,-2.414,-43.429,-179.810,5.628,148.935
C04997=1199.045,-2.664,-43.415,-179.813,5.628,148.936
C04998=1199.050,-2.914,-43.401,-179.814,5.628,148.937
C04999=1199.056,-3.163,-43.388,-179.817,5.627,148.937
C05000=1199.060,-3.413,-43.374,-179.819,5.627,148.938
C05001=1199.066,-3.662,-43.360,-179.822,5.626,148.939
C05002=1199.071,-3.912,-43.346,-179.825,5.626,148.939
C05003=1199.076,-4.161,-43.333,-179.827,5.625,148.940
C05004=1199.081,-4.410,-43.319,-179.830,5.624,148.940
C05005=1199.086,-4.661,-43.305,-179.832,5.624,148.941
C05006=1199.091,-4.910,-43.291,-179.834,5.624,148.942
C05007=1199.096,-5.159,-43.277,-179.837,5.624,148.943
C05008=1199.101,-5.409,-43.264,-179.840,5.623,148.943
C05009=1199.107,-5.658,-43.250,-179.842,5.622,148.944
C05010=1199.111,-5.908,-43.236,-179.844,5.622,148.944
C05011=1199.116,-6.158,-43.223,-179.847,5.621,148.945
C05012=1199.122,-6.407,-43.209,-179.850,5.621,148.946
C05013=1199.126,-6.657,-43.196,-179.852,5.621,148.946
C05014=1199.132,-6.906,-43.182,-179.854,5.621,148.947
C05015=1199.137,-7.156,-43.168,-179.857,5.620,148.948
C05016=1199.142,-7.406,-43.155,-179.859,5.619,148.948
C05017=1199.147,-7.655,-43.141,-179.862,5.619,148.949
C05018=1199.152,-7.905,-43.127,-179.865,5.618,148.950
C05019=1199.157,-8.154,-43.114,-179.867,5.619,148.950
C05020=1199.162,-8.404,-43.100,-179.869,5.618,148.951
C05021=1199.167,-8.654,-43.086,-179.871,5.617,148.952
C05022=1199.172,-8.903,-43.073,-179.874,5.617,148.952
C05023=1199.177,-9.153,-43.059,-179.877,5.616,148.953
C05024=1199.183,-9.402,-43.047,-179.879,5.616,148.954
C05025=1199.188,-9.652,-43.032,-179.882,5.616,148.954
C05026=1199.193,-9.902,-43.019,-179.884,5.616,148.955
C05027=1199.198,-10.151,-43.005,-179.886,5.615,148.955
C05028=1199.203,-10.401,-42.992,-179.889,5.614,148.956
C05029=1199.208,-10.650,-42.979,-179.892,5.614,148.957
C05030=1199.214,-10.900,-42.965,-179.894,5.614,148.958
C05031=1199.218,-11.149,-42.951,-179.897,5.613,148.958
C05032=1199.223,-11.399,-42.938,-179.899,5.613,148.959
C05033=1199.229,-11.648,-42.924,-179.901,5.613,148.959
C05034=1199.233,-11.898,-42.911,-179.904,5.612,148.960
C05035=1199.239,-12.147,-42.897,-179.907,5.612,148.961
C05036=1199.243,-12.397,-42.884,-179.909,5.611,148.961
C05037=1199.249,-12.647,-42.871,-179.912,5.611,148.962
C05038=1199.253,-12.897,-42.857,-179.913,5.611,148.963
C05039=1199.259,-13.146,-42.844,-179.916,5.610,148.963
C05040=1199.264,-13.396,-42.830,-179.919,5.610,148.964
C05041=1199.269,-13.645,-42.817,-179.921,5.609,148.965
C05042=1199.274,-13.895,-42.804,-179.924,5.609,148.965
C05043=1199.279,-14.144,-42.791,-179.926,5.609,148.966
C05044=1199.285,-14.395,-42.777,-179.928,5.608,148.967
C05045=1199.290,-14.644,-42.764,-179.931,5.608,148.967
C05046=1199.295,-14.893,-42.750,-179.934,5.607,148.968
C05047=1199.300,-15.143,-42.737,-179.936,5.607,148.969
C05048=1199.306,-15.392,-42.724,-179.939,5.606,148.969
C05049=1199.310,-15.642,-42.711,-179.941,5.607,148.970
C05050=1199.316,-15.892,-42.697,-179.943,5.606,148.970
C05051=1199.320,-16.142,-42.684,-179.946,5.605,148.971
C05052=1199.325,-16.390,-42.671,-179.948,5.605,148.972
C05053=1199.330,-16.641,-42.658,-179.951,5.604,148.973
C05054=1199.335,-16.890,-42.645,-179.953,5.605,148.973
C05055=1199.341,-17.140,-42.631,-179.956,5.604,148.974
C05056=1199.345,-17.389,-42.618,-179.958,5.603,148.974
C05057=1199.351,-17.639,-42.605,-179.961,5.603,148.975
C05058=1199.356,-17.889,-42.592,-179.963,5.602,148.976
C05059=1199.362,-18.138,-42.579,-179.965,5.603,148.976
C05060=1199.366,-18.388,-42.565,-179.968,5.602,148.977
C05061=1199.371,-18.637,-42.552,-179.971,5.602,148.978
C05062=1199.376,-18.887,-42.539,-179.973,5.601,148.978
C05063=1199.381,-19.137,-42.526,-179.976,5.600,148.979
C05064=1199.387,-19.386,-42.512,-179.978,5.601,148.980
C05065=1199.392,-19.636,-42.499,-179.980,5.600,148.980
C05066=1199.397,-19.885,-42.487,-179.983,5.600,148.981
C05067=1199.402,-20.135,-42.473,-179.986,5.599,148.982
C05068=1199.407,-20.385,-42.461,-179.988,5.598,148.982
C05069=1199.413,-20.634,-42.447,-179.990,5.599,148.983
C05070=1199.417,-20.884,-42.434,-179.993,5.598,148.984
C05071=1199.422,-21.133,-42.421,-179.995,5.598,148.984
C05072=1199.428,-21.383,-42.408,-179.998,5.597,148.985
C05073=1199.433,-21.633,-42.395,179.999,5.597,148.986
C05074=1199.438,-21.882,-42.382,179.998,5.597,148.986
C05075=1199.443,-22.132,-42.369,179.995,5.596,148.987
C05076=1199.448,-22.382,-42.356,179.993,5.596,148.988
C05077=1199.453,-22.631,-42.344,179.990,5.595,148.988
C05078=1199.459,-22.900,-42.329,179.987,5.595,148.989
C05079=1199.464,-23.170,-42.315,179.985,5.594,148.990
C05080=1199.470,-23.439,-42.301,179.983,5.595,148.990
C05081=1199.475,-23.709,-42.287,179.980,5.594,148.991
C05082=1199.481,-23.959,-42.274,179.977,5.594,148.992
C05083=1199.485,-24.209,-42.261,179.975,5.593,148.992
C05084=1199.491,-24.458,-42.249,179.972,5.593,148.993
C05085=1199.496,-24.708,-42.235,179.970,5.593,148.994
C05086=1199.501,-24.958,-42.222,179.968,5.592,148.994
C05087=1199.506,-25.207,-42.210,179.965,5.592,148.995
C05088=1199.511,-25.456,-42.197,179.962,5.591,148.996
C05089=1199.516,-25.707,-42.184,179.960,5.591,148.996
C05090=1199.522,-25.956,-42.171,179.958,5.591,148.997
C05091=1199.527,-26.205,-42.158,179.955,5.591,148.998
C05092=1199.531,-26.455,-42.146,179.953,5.590,148.998
C05093=1199.537,-26.705,-42.132,179.950,5.590,148.999
C05094=1199.542,-26.954,-42.120,179.948,5.590,149.000
C05095=1199.547,-27.204,-42.107,179.945,5.589,149.000
C05096=1199.552,-27.454,-42.094,179.943,5.589,149.001
C05097=1199.557,-27.703,-42.082,179.940,5.588,149.002
C05098=1199.563,-27.952,-42.068,179.938,5.588,149.002
C05099=1199.567,-28.203,-42.055,179.936,5.588,149.003
C05100=1199.572,-28.452,-42.043,179.933,5.587,149.004
C05101=1199.578,-28.701,-42.030,179.930,5.587,149.004
C05102=1199.583,-28.950,-42.018,179.928,5.587,149.005
C05103=1199.588,-29.201,-42.004,179.926,5.587,149.006
C05104=1199.593,-29.450,-41.991,179.924,5.586,149.006
C05105=1199.599,-29.700,-41.980,179.921,5.586,149.007
C05106=1199.603,-29.950,-41.967,179.918,5.585,149.008
C05107=1199.608,-30.199,-41.954,179.916,5.585,149.008
C05108=1199.613,-30.449,-41.941,179.913,5.585,149.009
C05109=1199.619,-30.698,-41.928,179.911,5.585,149.010
C05110=1199.624,-30.948,-41.916,179.909,5.584,149.010
C05111=1199.629,-31.198,-41.903,179.907,5.584,149.011
C05112=1199.634,-31.448,-41.891,179.904,5.584,149.012
C05113=1199.639,-31.697,-41.878,179.901,5.583,149.012
C05114=1199.644,-31.946,-41.866,179.899,5.583,149.013
C05115=1199.649,-32.196,-41.853,179.897,5.583,149.014
C05116=1199.654,-32.446,-41.840,179.894,5.582,149.014
C05117=1199.660,-32.696,-41.827,179.892,5.582,149.015
C05118=1199.665,-32.945,-41.815,179.889,5.581,149.016
C05119=1199.671,-33.194,-41.802,179.887,5.582,149.016
C05120=1199.675,-33.444,-41.789,179.884,5.581,149.017
C05121=1199.680,-33.694,-41.777,179.882,5.581,149.018
C05122=1199.686,-33.944,-41.765,179.880,5.581,149.018
C05123=1199.691,-34.193,-41.752,179.877,5.580,149.019
C05124=1199.696,-34.442,-41.740,179.875,5.580,149.019
C05125=1199.700,-34.692,-41.727,179.872,5.579,149.020
C05126=1199.706,-34.942,-41.715,179.870,5.580,149.021
C05127=1199.711,-35.192,-41.702,179.867,5.579,149.022
C05128=1199.716,-35.441,-41.690,179.865,5.578,149.022
C05129=1199.721,-35.691,-41.678,179.862,5.578,149.023
C05130=1199.727,-35.941,-41.664,179.860,5.578,149.023
C05131=1199.732,-36.191,-41.652,179.858,5.578,149.024
C05132=1199.737,-36.440,-41.640,179.855,5.577,149.025
C05133=1199.742,-36.690,-41.627,179.852,5.577,149.026
C05134=1199.748,-36.939,-41.614,179.851,5.577,149.026
C05135=1199.753,-37.189,-41.603,179.848,5.576,149.027
C05136=1199.758,-37.438,-41.590,179.845,5.576,149.027
C05137=1199.763,-37.688,-41.577,179.843,5.576,149.028
C05138=1199.768,-37.938,-41.565,179.841,5.576,149.029
C05139=1199.773,-38.188,-41.553,179.838,5.575,149.030
C05140=1199.778,-38.437,-41.540,179.836,5.574,149.030
C05141=1199.784,-38.687,-41.528,179.834,5.575,149.031
C05142=1199.789,-38.936,-41.515,179.831,5.574,149.031
C05143=1199.794,-39.186,-41.504,179.828,5.574,149.032
C05144=1199.799,-39.435,-41.491,179.826,5.574,149.033
C05145=1199.804,-39.685,-41.478,179.824,5.574,149.033
C05146=1199.809,-39.935,-41.467,179.822,5.573,149.034
C05147=1199.814,-40.184,-41.454,179.819,5.572,149.035
C05148=1199.819,-40.434,-41.442,179.817,5.573,149.035
C05149=1199.824,-40.684,-41.430,179.814,5.572,149.036
C05150=1199.830,-40.934,-41.418,179.811,5.572,149.037
C05151=1199.835,-41.183,-41.405,179.809,5.572,149.037
C05152=1199.840,-41.433,-41.393,179.807,5.571,149.038
C05153=1199.845,-41.682,-41.381,179.805,5.571,149.039
C05154=1199.851,-41.932,-41.369,179.802,5.570,149.039
C05155=1199.856,-42.181,-41.356,179.800,5.571,149.040
C05156=1199.861,-42.432,-41.344,179.797,5.570,149.041
C05157=1199.866,-42.681,-41.331,179.794,5.570,149.041
C05158=1199.871,-42.931,-41.320,179.793,5.570,149.042
C05159=1199.876,-43.180,-41.307,179.790,5.569,149.043
C05160=1199.881,-43.430,-41.296,179.788,5.569,149.043
C05161=1199.886,-43.680,-41.283,179.785,5.568,149.044
C05162=1199.892,-43.930,-41.271,179.783,5.569,149.045
C05163=1199.897,-44.179,-41.258,179.780,5.568,149.045
C05164=1199.902,-44.429,-41.247,179.778,5.567,149.046
C05165=1199.907,-44.678,-41.234,179.776,5.568,149.047
C05166=1199.912,-44.928,-41.223,179.773,5.567,149.047
C05167=1199.917,-45.177,-41.210,179.771,5.567,149.048
C05168=1199.923,-45.427,-41.198,179.768,5.567,149.049
C05169=1199.928,-45.677,-41.186,179.766,5.567,149.049
C05170=1199.933,-45.926,-41.174,179.764,5.566,149.050
C05171=1199.939,-46.176,-41.162,179.762,5.566,149.051
C05172=1199.943,-46.426,-41.150,179.759,5.566,149.051
C05173=1199.948,-46.675,-41.138,179.756,5.565,149.052
C05174=1199.954,-46.925,-41.126,179.754,5.565,149.053
C05175=1199.959,-47.174,-41.113,179.752,5.565,149.053
C05176=1199.964,-47.424,-41.102,179.749,5.565,149.054
C05177=1199.969,-47.674,-41.090,179.747,5.564,149.055
C05178=1199.974,-47.923,-41.078,179.745,5.564,149.055
C05179=1199.980,-48.173,-41.066,179.742,5.564,149.056
C05180=1199.985,-48.423,-41.054,179.739,5.564,149.057
C05181=1199.989,-48.672,-41.042,179.738,5.563,149.057
C05182=1199.996,-48.943,-41.028,179.735,5.563,149.058
C05183=1200.001,-49.213,-41.015,179.732,5.563,149.059
C05184=1200.007,-49.483,-41.003,179.729,5.563,149.059
C05185=1200.012,-49.753,-40.990,179.726,5.562,149.060
C05186=1200.017,-50.003,-40.978,179.725,5.562,149.061
C05187=1200.022,-50.253,-40.967,179.722,5.562,149.061
C05188=1200.027,-50.502,-40.954,179.720,5.561,149.062
C05189=1200.033,-50.752,-40.942,179.717,5.561,149.063
C05190=1200.037,-51.002,-40.931,179.715,5.561,149.063
C05191=1200.043,-51.252,-40.919,179.712,5.561,149.064
C05192=1200.049,-51.501,-40.907,179.711,5.561,149.065
C05193=1200.054,-51.750,-40.895,179.708,5.560,149.065
C05194=1200.059,-52.000,-40.884,179.705,5.560,149.066
C05195=1200.064,-52.250,-40.872,179.703,5.560,149.067
C05196=1200.070,-52.500,-40.860,179.700,5.560,149.067
C05197=1200.074,-52.749,-40.848,179.698,5.559,149.068
C05198=1200.079,-52.999,-40.836,179.696,5.559,149.069
C05199=1200.085,-53.248,-40.824,179.694,5.559,149.069
C05200=1200.089,-53.498,-40.813,179.691,5.558,149.070
C05201=1200.095,-53.748,-40.801,179.689,5.559,149.071
C05202=1200.100,-53.998,-40.789,179.686,5.558,149.071
C05203=1200.105,-54.247,-40.777,179.684,5.557,149.072
C05204=1200.110,-54.497,-40.765,179.682,5.558,149.073
C05205=1200.116,-54.747,-40.753,179.679,5.557,149.073
C05206=1200.121,-54.996,-40.742,179.677,5.557,149.074
C05207=1200.126,-55.246,-40.730,179.674,5.557,149.075
C05208=1200.131,-55.495,-40.719,179.672,5.557,149.075
C05209=1200.136,-55.745,-40.707,179.670,5.556,149.076
C05210=1200.142,-55.995,-40.695,179.668,5.556,149.077
C05211=1200.146,-56.244,-40.683,179.665,5.556,149.077
C05212=1200.152,-56.494,-40.671,179.662,5.555,149.078
C05213=1200.156,-56.744,-40.660,179.660,5.556,149.079
C05214=1200.162,-56.994,-40.648,179.658,5.555,149.079
C05215=1200.168,-57.243,-40.637,179.655,5.554,149.080
C05216=1200.173,-57.493,-40.625,179.653,5.555,149.081
C05217=1200.178,-57.742,-40.613,179.651,5.554,149.081
C05218=1200.183,-57.992,-40.602,179.648,5.554,149.082
C05219=1200.188,-58.242,-40.590,179.646,5.554,149.083
C05220=1200.193,-58.492,-40.579,179.644,5.553,149.083
C05221=1200.198,-58.742,-40.567,179.642,5.554,149.084
C05222=1200.203,-58.991,-40.556,179.639,5.553,149.085
C05223=1200.209,-59.240,-40.544,179.636,5.553,149.085
C05224=1200.214,-59.490,-40.533,179.634,5.553,149.086
C05225=1200.219,-59.740,-40.521,179.632,5.552,149.087
C05226=1200.224,-59.990,-40.509,179.629,5.552,149.087
C05227=1200.229,-60.240,-40.498,179.627,5.552,149.088
C05228=1200.235,-60.489,-40.486,179.624,5.552,149.089
C05229=1200.240,-60.738,-40.475,179.622,5.551,149.089
C05230=1200.245,-60.988,-40.463,179.620,5.551,149.090
C05231=1200.250,-61.238,-40.452,179.618,5.551,149.091
C05232=1200.255,-61.488,-40.440,179.615,5.551,149.091
C05233=1200.260,-61.738,-40.429,179.613,5.551,149.092
C05234=1200.266,-61.987,-40.417,179.610,5.550,149.093
C05235=1200.271,-62.236,-40.406,179.609,5.550,149.093
C05236=1200.276,-62.486,-40.394,179.606,5.550,149.094
C05237=1200.281,-62.737,-40.384,179.603,5.550,149.095
C05238=1200.286,-62.986,-40.372,179.601,5.550,149.095
C05239=1200.292,-63.235,-40.361,179.598,5.549,149.096
C05240=1200.297,-63.485,-40.349,179.596,5.549,149.096
C05241=1200.302,-63.735,-40.338,179.594,5.549,149.097
C05242=1200.307,-63.985,-40.326,179.592,5.549,149.098
C05243=1200.313,-64.234,-40.315,179.589,5.549,149.099
C05244=1200.318,-64.484,-40.303,179.587,5.549,149.099
C05245=1200.323,-64.734,-40.292,179.584,5.548,149.100
C05246=1200.328,-64.984,-40.281,179.583,5.548,149.100
C05247=1200.333,-65.233,-40.270,179.580,5.548,149.101
C05248=1200.339,-65.483,-40.258,179.577,5.547,149.102
C05249=1200.343,-65.732,-40.247,179.575,5.548,149.103
C05250=1200.349,-65.982,-40.235,179.572,5.547,149.103
C05251=1200.354,-66.232,-40.225,179.571,5.547,149.104
C05252=1200.359,-66.481,-40.214,179.568,5.547,149.104
C05253=1200.365,-66.731,-40.202,179.565,5.546,149.105
C05254=1200.369,-66.981,-40.190,179.563,5.547,149.106
C05255=1200.375,-67.230,-40.179,179.561,5.546,149.107
C05256=1200.380,-67.480,-40.168,179.559,5.545,149.107
C05257=1200.385,-67.730,-40.157,179.556,5.546,149.108
C05258=1200.390,-67.980,-40.145,179.554,5.545,149.108
C05259=1200.396,-68.229,-40.134,179.552,5.546,149.109
C05260=1200.401,-68.479,-40.124,179.549,5.545,149.110
C05261=1200.406,-68.729,-40.112,179.547,5.544,149.110
C05262=1200.411,-68.978,-40.101,179.545,5.545,149.111
C05263=1200.416,-69.228,-40.089,179.542,5.544,149.112
C05264=1200.422,-69.478,-40.078,179.540,5.545,149.112
C05265=1200.427,-69.727,-40.067,179.538,5.544,149.113
C05266=1200.432,-69.977,-40.056,179.535,5.543,149.114
C05267=1200.438,-70.227,-40.045,179.533,5.544,149.114
C05268=1200.442,-70.477,-40.034,179.530,5.543,149.115
C05269=1200.448,-70.726,-40.023,179.528,5.543,149.116
C05270=1200.453,-70.976,-40.012,179.526,5.543,149.116
C05271=1200.458,-71.226,-40.000,179.523,5.542,149.117
C05272=1200.463,-71.475,-39.989,179.521,5.543,149.118
C05273=1200.469,-71.725,-39.978,179.519,5.542,149.118
C05274=1200.474,-71.975,-39.967,179.516,5.542,149.119
C05275=1200.479,-72.224,-39.956,179.514,5.542,149.120
C05276=1200.485,-72.475,-39.945,179.512,5.542,149.120
C05277=1200.490,-72.723,-39.934,179.510,5.542,149.121
C05278=1200.495,-72.974,-39.923,179.507,5.541,149.122
C05279=1200.500,-73.223,-39.912,179.504,5.541,149.122
C05280=1200.506,-73.473,-39.900,179.503,5.541,149.123
C05281=1200.511,-73.723,-39.890,179.500,5.541,149.124
C05282=1200.515,-73.972,-39.879,179.498,5.541,149.124
C05283=1200.521,-74.222,-39.868,179.495,5.541,149.125
C05284=1200.526,-74.472,-39.857,179.493,5.540,149.125
C05285=1200.531,-74.722,-39.845,179.491,5.540,149.126
C05286=1200.538,-74.992,-39.834,179.488,5.540,149.127
C05287=1200.543,-75.263,-39.822,179.486,5.539,149.128
C05288=1200.549,-75.533,-39.811,179.484,5.540,149.128
C05289=1200.554,-75.804,-39.798,179.481,5.539,149.129
C05290=1200.559,-76.054,-39.787,179.478,5.539,149.130
C05291=1200.565,-76.304,-39.777,179.476,5.539,149.130
C05292=1200.569,-76.553,-39.765,179.474,5.539,149.131
C05293=1200.576,-76.803,-39.755,179.472,5.539,149.132
C05294=1200.580,-77.053,-39.743,179.469,5.538,149.132
C05295=1200.585,-77.303,-39.733,179.467,5.538,149.133
C05296=1200.591,-77.552,-39.722,179.465,5.538,149.134
C05297=1200.596,-77.802,-39.711,179.462,5.538,149.134
C05298=1200.601,-78.051,-39.700,179.460,5.538,149.135
C05299=1200.607,-78.302,-39.689,179.458,5.537,149.136
C05300=1200.612,-78.552,-39.679,179.455,5.538,149.136
C05301=1200.617,-78.801,-39.668,179.453,5.537,149.137
C05302=1200.622,-79.051,-39.657,179.451,5.536,149.138
C05303=1200.627,-79.300,-39.646,179.449,5.537,149.138
C05304=1200.632,-79.550,-39.636,179.446,5.536,149.139
C05305=1200.638,-79.799,-39.625,179.444,5.537,149.140
C05306=1200.643,-80.050,-39.614,179.441,5.536,149.140
C05307=1200.649,-80.299,-39.603,179.439,5.536,149.141
C05308=1200.654,-80.549,-39.592,179.437,5.536,149.142
C05309=1200.659,-80.799,-39.581,179.434,5.535,149.142
C05310=1200.664,-81.048,-39.571,179.432,5.536,149.143
C05311=1200.669,-81.298,-39.560,179.430,5.535,149.143
C05312=1200.674,-81.548,-39.550,179.428,5.535,149.144
C05313=1200.679,-81.797,-39.538,179.425,5.535,149.145
C05314=1200.685,-82.047,-39.528,179.422,5.535,149.146
C05315=1200.690,-82.297,-39.518,179.421,5.535,149.146
C05316=1200.696,-82.546,-39.506,179.418,5.534,149.147
C05317=1200.701,-82.797,-39.496,179.416,5.534,149.147
C05318=1200.706,-83.046,-39.485,179.413,5.534,149.148
C05319=1200.711,-83.296,-39.474,179.412,5.534,149.149
C05320=1200.717,-83.545,-39.464,179.409,5.534,149.149
C05321=1200.722,-83.796,-39.453,179.407,5.533,149.150
C05322=1200.727,-84.045,-39.442,179.404,5.534,149.151
C05323=1200.732,-84.295,-39.432,179.402,5.533,149.152
C05324=1200.738,-84.544,-39.422,179.400,5.533,149.152
C05325=1200.742,-84.794,-39.410,179.397,5.533,149.153
C05326=1200.748,-85.043,-39.400,179.395,5.533,149.153
C05327=1200.753,-85.294,-39.390,179.393,5.533,149.154
C05328=1200.758,-85.543,-39.379,179.391,5.532,149.155
C05329=1200.763,-85.793,-39.368,179.388,5.532,149.155
C05330=1200.769,-86.042,-39.358,179.386,5.532,149.156
C05331=1200.774,-86.293,-39.347,179.384,5.532,149.157
C05332=1200.779,-86.542,-39.337,179.382,5.531,149.157
C05333=1200.784,-86.792,-39.326,179.379,5.532,149.158
C05334=1200.790,-87.041,-39.316,179.377,5.531,149.159
C05335=1200.795,-87.292,-39.305,179.375,5.532,149.159
C05336=1200.800,-87.541,-39.295,179.372,5.531,149.160
C05337=1200.805,-87.791,-39.283,179.370,5.531,149.161
C05338=1200.810,-88.040,-39.273,179.368,5.531,149.161
C05339=1200.816,-88.290,-39.263,179.365,5.530,149.162
C05340=1200.821,-88.540,-39.252,179.363,5.530,149.162
C05341=1200.827,-88.790,-39.242,179.361,5.530,149.163
C05342=1200.831,-89.040,-39.232,179.359,5.530,149.164
C05343=1200.836,-89.289,-39.221,179.356,5.530,149.165
C05344=1200.841,-89.539,-39.211,179.354,5.530,149.165
C05345=1200.847,-89.788,-39.201,179.352,5.530,149.166
C05346=1200.852,-90.038,-39.190,179.349,5.529,149.166
C05347=1200.857,-90.288,-39.180,179.347,5.530,149.167
C05348=1200.863,-90.538,-39.170,179.345,5.529,149.168
C05349=1200.868,-90.788,-39.159,179.343,5.529,149.168
C05350=1200.873,-91.037,-39.148,179.340,5.529,149.169
C05351=1200.878,-91.287,-39.138,179.338,5.529,149.170
C05352=1200.884,-91.537,-39.127,179.336,5.528,149.170
C05353=1200.889,-91.786,-39.118,179.334,5.529,149.171
C05354=1200.894,-92.036,-39.107,179.331,5.528,149.172
C05355=1200.899,-92.286,-39.097,179.329,5.528,149.172
C05356=1200.904,-92.536,-39.086,179.327,5.528,149.173
C05357=1200.910,-92.785,-39.076,179.324,5.527,149.174
C05358=1200.916,-93.035,-39.066,179.322,5.528,149.174
C05359=1200.921,-93.285,-39.055,179.320,5.527,149.175
C05360=1200.926,-93.535,-39.045,179.318,5.527,149.176
C05361=1200.931,-93.784,-39.036,179.315,5.527,149.176
C05362=1200.936,-94.034,-39.025,179.313,5.527,149.177
C05363=1200.942,-94.284,-39.015,179.311,5.527,149.177
C05364=1200.947,-94.533,-39.005,179.309,5.527,149.178
C05365=1200.952,-94.784,-38.994,179.306,5.526,149.179
C05366=1200.958,-95.033,-38.984,179.304,5.527,149.180
C05367=1200.962,-95.283,-38.974,179.302,5.526,149.180
C05368=1200.968,-95.533,-38.964,179.300,5.526,149.181
C05369=1200.973,-95.782,-38.953,179.297,5.526,149.181
C05370=1200.978,-96.032,-38.943,179.295,5.526,149.182
C05371=1200.984,-96.282,-38.933,179.293,5.526,149.183
C05372=1200.989,-96.531,-38.923,179.290,5.525,149.183
C05373=1200.994,-96.781,-38.912,179.288,5.526,149.184
C05374=1200.999,-97.031,-38.902,179.286,5.525,149.185
C05375=1201.005,-97.280,-38.892,179.284,5.525,149.185
C05376=1201.010,-97.531,-38.881,179.281,5.525,149.186
C05377=1201.015,-97.780,-38.872,179.279,5.525,149.187
C05378=1201.020,-98.029,-38.862,179.277,5.524,149.187
C05379=1201.026,-98.279,-38.851,179.275,5.525,149.188
C05380=1201.031,-98.529,-38.841,179.272,5.524,149.189
C05381=1201.036,-98.779,-38.831,179.270,5.524,149.189
C05382=1201.041,-99.028,-38.821,179.268,5.524,149.190
C05383=1201.047,-99.279,-38.811,179.266,5.524,149.191
C05384=1201.052,-99.528,-38.801,179.263,5.524,149.191
C05385=1201.057,-99.778,-38.791,179.261,5.524,149.192
C05386=1201.062,-100.028,-38.781,179.259,5.523,149.192
C05387=1201.068,-100.277,-38.771,179.257,5.524,149.193
C05388=1201.073,-100.527,-38.760,179.254,5.523,149.194
C05389=1201.078,-100.776,-38.751,179.252,5.523,149.194
C05390=1201.084,-101.048,-38.740,179.250,5.523,149.195
C05391=1201.090,-101.320,-38.729,179.247,5.523,149.196
C05392=1201.095,-101.591,-38.718,179.245,5.523,149.196
C05393=1201.101,-101.862,-38.707,179.242,5.523,149.197
C05394=1201.106,-102.113,-38.698,179.239,5.522,149.198
C05395=1201.112,-102.362,-38.687,179.238,5.522,149.198
C05396=1201.117,-102.612,-38.677,179.235,5.522,149.199
C05397=1201.122,-102.861,-38.668,179.233,5.522,149.200
C05398=1201.127,-103.111,-38.657,179.231,5.521,149.200
C05399=1201.133,-103.361,-38.647,179.229,5.522,149.201
C05400=1201.138,-103.610,-38.638,179.226,5.521,149.202
C05401=1201.143,-103.860,-38.628,179.225,5.521,149.202
C05402=1201.148,-104.110,-38.617,179.222,5.521,149.203
C05403=1201.154,-104.360,-38.608,179.220,5.521,149.204
C05404=1201.159,-104.610,-38.598,179.217,5.521,149.204
C05405=1201.165,-104.859,-38.588,179.216,5.521,149.205
C05406=1201.169,-105.109,-38.578,179.213,5.521,149.206
C05407=1201.175,-105.359,-38.568,179.211,5.521,149.206
C05408=1201.180,-105.609,-38.559,179.209,5.520,149.207
C05409=1201.185,-105.858,-38.548,179.206,5.521,149.207
C05410=1201.191,-106.108,-38.539,179.204,5.520,149.208
C05411=1201.196,-106.358,-38.529,179.202,5.520,149.209
C05412=1201.201,-106.608,-38.519,179.200,5.520,149.209
C05413=1201.206,-106.857,-38.509,179.197,5.520,149.210
C05414=1201.212,-107.107,-38.500,179.195,5.519,149.211
C05415=1201.217,-107.357,-38.489,179.193,5.520,149.211
C05416=1201.222,-107.607,-38.479,179.190,5.519,149.212
C05417=1201.228,-107.857,-38.470,179.188,5.520,149.213
C05418=1201.232,-108.106,-38.460,179.186,5.519,149.213
C05419=1201.238,-108.356,-38.450,179.184,5.519,149.214
C05420=1201.243,-108.605,-38.441,179.181,5.519,149.215
C05421=1201.249,-108.855,-38.431,179.180,5.519,149.215
C05422=1201.254,-109.106,-38.421,179.177,5.518,149.216
C05423=1201.259,-109.355,-38.412,179.175,5.519,149.217
C05424=1201.265,-109.605,-38.401,179.173,5.518,149.217
C05425=1201.270,-109.854,-38.392,179.171,5.518,149.218
C05426=1201.275,-110.104,-38.382,179.168,5.518,149.218
C05427=1201.281,-110.354,-38.373,179.167,5.518,149.219
C05428=1201.286,-110.604,-38.363,179.164,5.518,149.220
C05429=1201.290,-110.853,-38.353,179.162,5.518,149.220
C05430=1201.296,-111.103,-38.344,179.160,5.517,149.221
C05431=1201.301,-111.353,-38.334,179.157,5.518,149.222
C05432=1201.307,-111.603,-38.325,179.155,5.517,149.222
C05433=1201.312,-111.852,-38.315,179.153,5.517,149.223
C05434=1201.318,-112.102,-38.305,179.151,5.517,149.223
C05435=1201.322,-112.352,-38.295,179.148,5.517,149.224
C05436=1201.328,-112.602,-38.285,179.146,5.516,149.225
C05437=1201.333,-112.852,-38.276,179.144,5.517,149.225
C05438=1201.338,-113.101,-38.266,179.141,5.516,149.226
C05439=1201.344,-113.351,-38.257,179.140,5.516,149.227
C05440=1201.349,-113.601,-38.247,179.137,5.516,149.227
C05441=1201.354,-113.850,-38.238,179.135,5.516,149.228
C05442=1201.360,-114.100,-38.228,179.133,5.516,149.229
C05443=1201.365,-114.350,-38.219,179.131,5.516,149.229
C05444=1201.370,-114.600,-38.208,179.128,5.516,149.230
C05445=1201.375,-114.850,-38.200,179.127,5.516,149.230
C05446=1201.380,-115.100,-38.191,179.124,5.515,149.231
C05447=1201.386,-115.349,-38.180,179.122,5.516,149.232
C05448=1201.391,-115.599,-38.172,179.120,5.515,149.232
C05449=1201.397,-115.849,-38.161,179.118,5.515,149.233
C05450=1201.402,-116.099,-38.152,179.115,5.515,149.234
C05451=1201.408,-116.348,-38.142,179.113,5.515,149.234
C05452=1201.413,-116.598,-38.133,179.111,5.514,149.235
C05453=1201.418,-116.847,-38.124,179.109,5.514,149.235
C05454=1201.424,-117.097,-38.114,179.106,5.514,149.236
C05455=1201.429,-117.347,-38.105,179.104,5.514,149.237
C05456=1201.434,-117.597,-38.095,179.102,5.514,149.237
C05457=1201.439,-117.847,-38.086,179.100,5.514,149.238
C05458=1201.444,-118.096,-38.076,179.098,5.514,149.239
C05459=1201.450,-118.347,-38.067,179.096,5.514,149.239
C05460=1201.455,-118.596,-38.058,179.094,5.514,149.240
C05461=1201.460,-118.846,-38.048,179.091,5.514,149.241
C05462=1201.466,-119.096,-38.039,179.089,5.514,149.241
C05463=1201.471,-119.346,-38.030,179.087,5.513,149.242
C05464=1201.476,-119.595,-38.020,179.084,5.514,149.243
C05465=1201.482,-119.845,-38.011,179.082,5.513,149.243
C05466=1201.487,-120.095,-38.002,179.080,5.513,149.244
C05467=1201.492,-120.344,-37.992,179.078,5.513,149.244
C05468=1201.497,-120.594,-37.983,179.076,5.513,149.245
C05469=1201.503,-120.844,-37.974,179.073,5.513,149.246
C05470=1201.507,-121.093,-37.964,179.072,5.513,149.246
C05471=1201.513,-121.344,-37.955,179.069,5.512,149.247
C05472=1201.519,-121.593,-37.946,179.067,5.513,149.248
C05473=1201.523,-121.843,-37.936,179.065,5.512,149.248
C05474=1201.529,-122.093,-37.927,179.063,5.512,149.249
C05475=1201.534,-122.343,-37.918,179.060,5.511,149.249
C05476=1201.540,-122.593,-37.909,179.058,5.512,149.250
C05477=1201.545,-122.842,-37.899,179.056,5.512,149.251
C05478=1201.550,-123.092,-37.890,179.054,5.511,149.251
C05479=1201.556,-123.342,-37.881,179.052,5.512,149.252
C05480=1201.560,-123.591,-37.871,179.049,5.511,149.253
C05481=1201.566,-123.841,-37.862,179.048,5.511,149.253
C05482=1201.571,-124.091,-37.853,179.045,5.511,149.254
C05483=1201.577,-124.341,-37.844,179.043,5.511,149.254
C05484=1201.582,-124.591,-37.835,179.041,5.511,149.255
C05485=1201.587,-124.840,-37.825,179.039,5.511,149.256
C05486=1201.593,-125.090,-37.816,179.036,5.510,149.256
C05487=1201.598,-125.340,-37.807,179.034,5.511,149.257
C05488=1201.603,-125.590,-37.798,179.032,5.510,149.258
